RoboDK station: DK_mettoolswitch_en_meerderematen.rdk

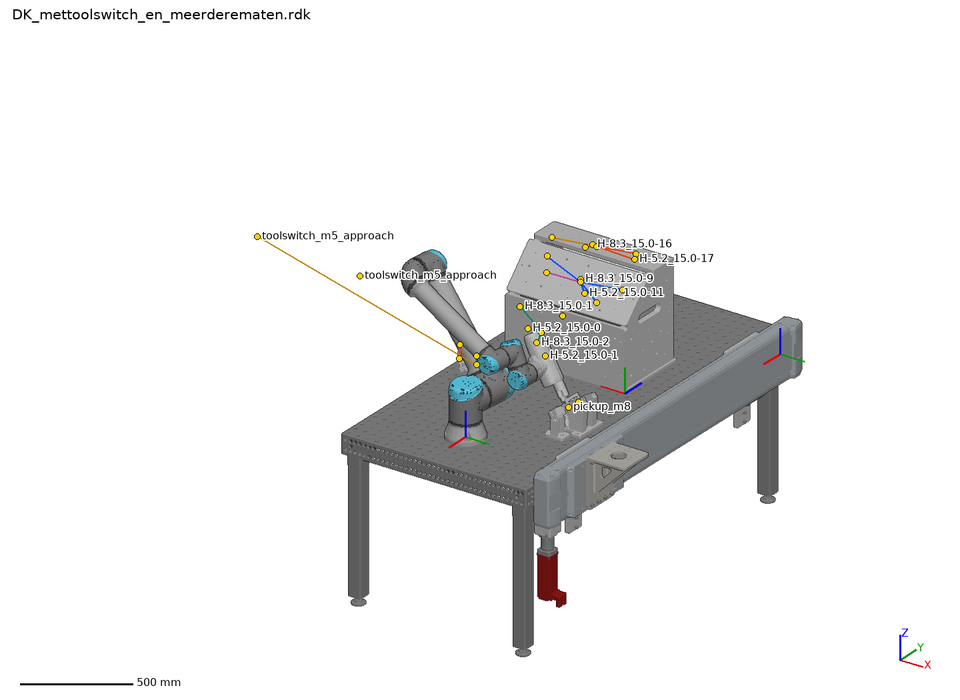
[picture v0: the station drawn from its stored meshes, robots at their saved joint values, targets as dots, program paths as lines]
Station DK_mettoolswitch_en_meerderematen (saved by RoboDK 5.9.0). Poses are relative to the parent item; angles as X-Y-Z fixed-axis rotations.
Station parameters (name, value as stored): CollisionFreePlanner, UR10e, CollisionFreePlanner-Rob UR10e, CollisionFreePlanner-Rob My Mechanism, CollisionFreePlanner-Rob Lineaire rail
  - object Lineaire Rail at (0, 0, 0) mm, size 171.1 x 1963 x 635.1 mm
  - object Cobot Carraige at (0, 0, 0) mm, size 240 x 425 x 269.5 mm
  - object Lastafel at (0, 0, 0) mm, size 1021.8 x 2000 x 842 mm
  - frame UR10e Base at (-522.25, 125.5, 70) mm, rotated rx 0 ry 0 rz -90 deg
    - robot UR10e: 6 axes, payload 10 kg, reach 1300 mm, repeatability 0.05 mm, weight 28.9 kg
        modified DH rows (alpha deg, a mm, theta deg, d mm): 0, 0, 0, 180.7; 90, 0, 180, 0; 0, 612.6, 0, 0; 0, 571.335, 0, 174.15; -90, 0, 0, 119.85; 90, 0, 180, 116.55
        joint limits [-100, -150, -30, -360, -360, -360] to [40, 0, 180, 360, 360, 360]; home [30.872, -95.296, 116.362, -22.187, 121.11, 179.827]; saved at [-96.274, -127.936, 155.823, 308.08, -8.026, -97.355]
      - tool schroevendraaier all in met nieuw kopstuk en tool, TCP at (220, -1, 100.6) mm, rotated rx 0 ry -90 rz 180 deg, size 86.2 x 139.7 x 345.9 mm, geometry from schroevendraaier all in met nieuw kopstuk en tool.STEP
  - frame Lineaire rail  Base at (218.83, 1501.27, 137) mm, rotated rx 0 ry 0 rz -90 deg
    - robot Lineaire rail: 1 axes
        modified DH rows (alpha deg, a mm, theta deg, d mm): 0, 0, 0, 0 linear
        base shift (0, 0, 0) mm, rotated rx 0 ry 90 rz 0 deg
        joint limits [-1248] to [-1248]; home [0]; saved at [-1248]
  - frame CSV Frame at (-220, 926.5, 50) mm, rotated rx 90 ry 0 rz 180 deg
    - object Test object at (0, 0, 0) mm, size 650 x 517 x 400 mm, geometry from Test object.STEP
    - object Toolswitch M5 M8 M12 (1) at (725, 0, -238) mm, size 112.6 x 60.1 x 126.6 mm, geometry from Toolswitch M5 M8 M12 (1).STEP
    - object Festo pneumatisch klem-1 at (22.5, 67, -437.5) mm, rotated rx 0 ry -90 rz -30 deg, size 249.3 x 187.1 x 198.8 mm, geometry from Festo pneumatisch klem-1.STEP
    - target pickup_m8 (Cartesian target) at (-3.8, 107.38, -439.03) mm, rotated rx 130.69 ry -86.57 rz -71.9 deg; joints [-96.274, -127.938, 155.828, 308.074, -8.028, -97.355] of UR10e
    - target pickup_m5 (Cartesian target) at (-2.38, 103.06, -363.09) mm, rotated rx 130.69 ry -86.57 rz -71.9 deg; joints [-75.565, -105.059, 145.828, -26.927, 13.754, -134.641] of UR10e
    - target H-8.3_15.0-1 (Cartesian target) at (577.65, 261.77, 15) mm; joints [-8.85, -55.871, 121.874, 293.989, -8.849, -179.992] of UR10e
    - target H-8.3_15.0-2 (Cartesian target) at (487.08, 107.86, 15) mm; joints [-11.324, -73.615, 119.159, 314.45, -11.322, -179.994] of UR10e
    - target H-8.3_15.0-9 (Cartesian target) at (325.68, 421.98, 122.91) mm, rotated rx 45 ry 0 rz 0 deg; joints [-39.434, -56.578, 53.669, 2.907, -39.433, -134.999] of UR10e
    - target H-8.3_15.0-11 (Cartesian target) at (502.06, 411.39, 112.31) mm, rotated rx 45 ry 0 rz 0 deg; joints [-28.45, -75.722, 93.025, -17.305, -28.449, -134.998] of UR10e
    - target H-8.3_15.0-16 (Cartesian target) at (391.06, 502, 308.3) mm, rotated rx -90 ry -83.43 rz 180 deg; joints [-3.833, -57.961, 69.865, -191.904, -92.74, -270.001] of UR10e
    - target H-8.3_15.0-17 (Cartesian target) at (577.65, 502, 262.67) mm, rotated rx 90 ry -81.14 rz 0 deg; joints [4.596, -59.728, 72.637, -192.908, -85.739, 89.999] of UR10e
    - target H-5.2_15.0-0 (Cartesian target) at (535.43, 162.34, 15) mm; joints [-96.274, -127.938, 155.828, 308.074, -8.028, -97.355] of UR10e
    - target H-5.2_15.0-1 (Cartesian target) at (442.81, 53.38, 15) mm; joints [-15.442, -65.401, 121.917, 303.479, -15.441, -179.996] of UR10e
    - target H-5.2_15.0-2 (Cartesian target) at (346.79, 277.43, 15) mm; joints [-24.169, -54.535, 121.923, 292.609, -24.168, -179.997] of UR10e
    - target H-5.2_15.0-10 (Cartesian target) at (534.75, 462.43, 163.36) mm, rotated rx 45 ry 0 rz 0 deg; joints [-11.699, -75.041, 88.001, 347.035, -11.697, -134.994] of UR10e
    - target H-5.2_15.0-11 (Cartesian target) at (278.01, 382.49, 83.42) mm, rotated rx 45 ry 0 rz 0 deg; joints [-11.354, -69.052, 72.632, 356.413, -11.353, -134.994] of UR10e
    - target H-5.2_15.0-12 (Cartesian target) at (103, 429.68, 130.61) mm, rotated rx 45 ry 0 rz 0 deg; joints [-31.461, -71.951, 84.687, 347.262, -31.46, -134.998] of UR10e
    - target H-5.2_15.0-15 (Cartesian target) at (197.65, 365.16, 66.09) mm, rotated rx 45 ry 0 rz 0 deg; joints [-20.089, -72.116, 80.974, 351.138, -20.088, -134.997] of UR10e
    - target H-5.2_15.0-16 (Cartesian target) at (178.59, 502, 342.35) mm, rotated rx -90 ry -85.2 rz -180 deg; joints [-17.19, -54.726, 64.672, 170.054, -77.607, -270.001] of UR10e
    - target H-5.2_15.0-17 (Cartesian target) at (151.35, 502, 290.59) mm, rotated rx 90 ry -89.07 rz 0 deg; joints [-21.263, -59.263, 71.911, 167.352, -67.807, -270.001] of UR10e
    - target H-5.2_15.0-19 (Cartesian target) at (403.31, 502, 268.12) mm, rotated rx 90 ry -77.85 rz 0 deg; joints [-7.94, -62.095, 76.272, 165.823, -69.913, -270.001] of UR10e
    - target toolswitch_m5_approach (Cartesian target) at (678.21, 67.52, -177.75) mm, rotated rx 90.07 ry 0.02 rz 0 deg; joints [-1.416, -72.071, 113.252, 318.849, -1.438, -89.956] of UR10e
      - target toolswitch_m5_approach (Cartesian target) at (678.21, 67.52, -177.75) mm, rotated rx 90.07 ry 0.02 rz 0 deg; joints [-1.416, -72.071, 113.252, 318.849, -1.438, -89.956] of UR10e
      - target toolswitch_m5_approach (Cartesian target) at (678.21, 67.52, -177.75) mm, rotated rx 90.07 ry 0.02 rz 0 deg; joints [-1.416, -72.071, 113.252, 318.849, -1.438, -89.956] of UR10e
        - target toolswitch_m5_approach (Cartesian target) at (678.21, 67.52, -177.75) mm, rotated rx 90.07 ry 0.02 rz 0 deg; joints [-1.416, -72.071, 113.252, 318.849, -1.438, -89.956] of UR10e
    - target toolswitch_m5 (Cartesian target) at (678.21, 21.65, -177.28) mm, rotated rx 90.14 ry 0.02 rz 0 deg; joints [-1.415, -68.774, 114.67, 314.195, -1.435, -89.952] of UR10e
    - target toolswitch_m8_approach (Cartesian target) at (769.79, 96.06, -177.07) mm, rotated rx 90.13 ry 0.05 rz -0.01 deg; joints [6.859, -71.505, 108.744, 322.817, 6.815, -89.924] of UR10e
    - target toolswitch_m8 (Cartesian target) at (769.77, 26.3, -177.21) mm, rotated rx 90.12 ry 0.04 rz 0 deg; joints [6.858, -66.989, 111.2, 315.836, 6.816, -89.924] of UR10e
    - target Face_Target_0 (Cartesian target) at (462.22, 165.4, 15) mm; joints [-91.475, -122.804, 153.527, 230.74, -2.975, -106.105] of UR10e
    - target Face_Target_1 (Cartesian target) at (318.87, 413.79, 114.72) mm, rotated rx 45 ry 0 rz 0 deg; joints [-91.475, -122.804, 153.527, 230.74, -2.975, -106.105] of UR10e
    - target Face_Target_2 (Cartesian target) at (364.5, 502, 302.51) mm, rotated rx -90 ry -83.43 rz 180 deg; joints [-91.475, -122.804, 153.527, 230.74, -2.975, -106.105] of UR10e
  - Python program csv_importer (listed below)
  - Python program csv_importernewest (listed below)
  - Python program Make_approaches_paths (listed below)
  - Python program TargetFixer (listed below)
  - Python program generatefaceapproaches (listed below)
  - Python program Addmoveshanktoprog (listed below)
  - Python program importerTest (listed below)
  - Python program Create measurements 3DOF (listed below)
  - Python program Prog11 (listed below)
  - Python program ProgramGenerator (listed below)
    - Python program ProgramGenerator (listed below)
  - program pickupm5Totoolswitchm8approach (13 instructions, listed below)
  - program Program_Main_Combined_met (7 instructions, listed below)
  - program Program_Main_Combined_met (13 instructions, listed below)
  - program Program_Main_Combined_met (2 instructions, listed below)
  - program Prog43 (10 instructions, listed below)
  - program pickupm8Totoolswitchm8 (12 instructions, listed below)
  - program toolswitchm8Topickupm8 (12 instructions, listed below)
  - program pickupm5Totoolswitchm5 (10 instructions, listed below)
  - program toolswitchm5Topickupm5 (10 instructions, listed below)
  - program FaceTarget0ToPickupm8 (6 instructions, listed below)
  - program Pickupm8ToFaceTarget0 (6 instructions, listed below)
  - program FaceTarget1ToPickupm8 (8 instructions, listed below)
  - program Pickupm8ToFaceTarget1 (8 instructions, listed below)
  - program FaceTarget2ToPickupm8 (15 instructions, listed below)
  - program Pickupm8ToFaceTarget2 (14 instructions, listed below)
  - program Program_Face_0_m8 (17 instructions, listed below)
  - program Program_Face_1_m8 (16 instructions, listed below)
  - program Program_Face_2_m8 (15 instructions, listed below)
  - program FaceTarget0ToPickupm5 (12 instructions, listed below)
  - program Pickupm5ToFaceTarget0 (12 instructions, listed below)
  - program FaceTarget1ToPickupm5 (12 instructions, listed below)
  - program Pickupm5ToFaceTarget1 (12 instructions, listed below)
  - program FaceTarget2ToPickupm5 (9 instructions, listed below)
  - program Pickupm5ToFaceTarget2 (8 instructions, listed below)
  - program Program_Face_0_m5 (6 instructions, listed below)
  - program Program_Face_1_m5 (33 instructions, listed below)
  - program Program_Face_2_m5 (25 instructions, listed below)
  - program Program_Main_m8 (5 instructions, listed below)
  - program Program_Main_m5 (5 instructions, listed below)
  - program pickupm8Totoolswitchm8approach (16 instructions, listed below)
  - program toolswitchm8approachTopickupm8 (16 instructions, listed below)
  - program Tool_Pickup_m8 (5 instructions, listed below)
  - program Tool_Dropoff_m8 (5 instructions, listed below)
  - program pickupm5Totoolswitchm5approach (12 instructions, listed below)
  - program toolswitchm5approachTopickupm5 (12 instructions, listed below)
  - program Tool_Pickup_m5 (6 instructions, listed below)
  - program Tool_Dropoff_m5 (5 instructions, listed below)
  - program Program_Main_Combined (8 instructions, listed below)
  - program toolswitchm5approachTopickupm8 (13 instructions, listed below)
  - program pickupm8Totoolswitchm5approach (13 instructions, listed below)
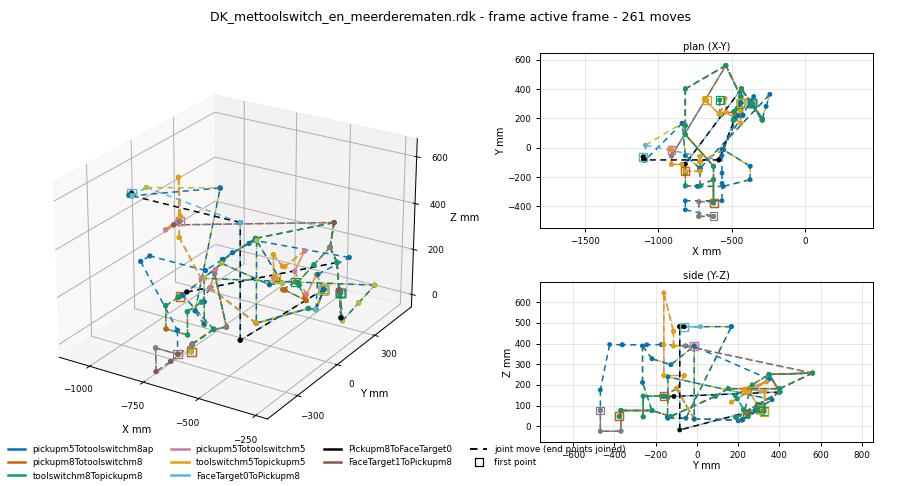
[picture p0: tool path of DK_mettoolswitch_en_meerderematen.rdk in frame active frame, 261 of 322 moves have a stored position in this frame; points joined in program order, loops and branches not executed]
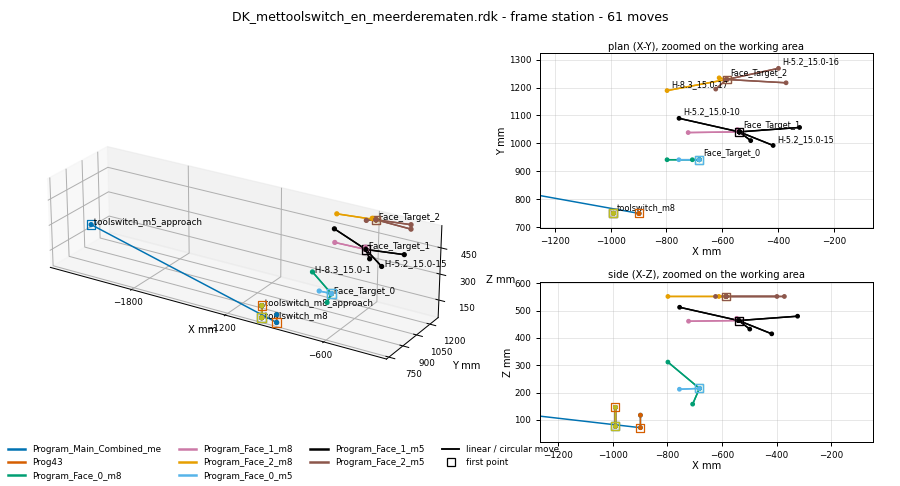
[picture p1: tool path of DK_mettoolswitch_en_meerderematen.rdk in frame station, 61 of 322 moves have a stored position in this frame; points joined in program order, loops and branches not executed]

--- Python program csv_importer ---
# This macro can load CSV files from Denso programs in RoboDK.
# Supported types of files are:
#  1-Tool data : Tool.csv
#  2-Work object data: Work.csv
#  3-Target data: P_Var.csv
# This macro can also filter a given targets file

# Type help("robodk.robolink") or help("robodk.robomath") for more information
# Press F5 to run the script
# Visit: http://www.robodk.com/doc/PythonAPI/
# For RoboDK API documentation

import os
import datetime

import tkinter as tk
from tkinter import messagebox

from robodk.robolink import *  # API to communicate with RoboDK
from robodk.robomath import *  # Robot toolbox
from robodk.robodialogs import *
from robodk.robofileio import *
import robodk.robolinkutils as RDKutils

DEBUG = False

debuglist = []

# Start communication with RoboDK
RDK = Robolink()

# Ask the user to select the robot
ROBOT = RDK.ItemUserPick('Select a robot', ITEM_TYPE_ROBOT)

# Check if the user selected a robot
if not ROBOT.Valid():
    quit()


# Ask the user to select a reference frame and get the active tool
BASE = ROBOT.Parent()
#BASE = RDK.Item('UR10e Base', ITEM_TYPE_FRAME)
#BASE = RDK.ItemUserPick('Select robot base frame', ITEM_TYPE_FRAME)
FRAME = RDK.ItemUserPick('Reference Frame', ITEM_TYPE_FRAME)
FRAMEPOSE = RDKutils.getPoseWrt(FRAME, BASE) #frame pose wrt robot base
TOOL = ROBOT.getLink(ITEM_TYPE_TOOL)
TOOLPOSE = RDKutils.getPoseWrt(TOOL, TOOL.Parent()) #tool pose wrt robot flange

if not FRAME.Valid() or not TOOL.Valid():
    raise Exception("Select appropriate FRAME and TOOL references")


# Function to convert XYZWPR to a pose
# Important! Specify the order of rotation
def xyzwpr_to_pose(xyzwpr):
    x, y, z, rx, ry, rz = xyzwpr
    return point_Zaxis_2_pose([x, y, z], [-rx, -ry, -rz])



# csv_file = 'C:/Users/Albert/Desktop/Var_P.csv'
csv_file = getOpenFileName(RDK.getParam('PATH_OPENSTATION'))

# Specify file codec
codec = 'utf-8'  #'ISO-8859-1'

def mirror_target(xyzwpr):
    """
    Mirrors the target position and adjusts the rotation.
    Assumes the wall is aligned with the YZ plane (mirroring the X coordinate).
    """
    x, y, z, rx, ry, rz = xyzwpr

    # Mirror the position (reflect across the YZ plane)
    x_mirrored = x  # Negate the X coordinate
    y_mirrored = y   # Keep Y and Z the same
    z_mirrored = z

    # Adjust the rotation (flip RX and RZ)
    rx_mirrored = rx  # Negate RX
    ry_mirrored = ry   # Keep RY the same
    rz_mirrored = -rz  # Negate RZ

    return [x_mirrored, y_mirrored, z_mirrored, rx_mirrored, ry_mirrored, rz_mirrored]

def load_targets(strfile):
    csvdata = LoadList(strfile, ',', codec)
    poses = []
    idxs = []
    for i in range(0, len(csvdata)):
        x, y, z, rx, ry, rz = csvdata[i][0:6]

        # Mirror the target
        x_mirrored, y_mirrored, z_mirrored, rx_mirrored, ry_mirrored, rz_mirrored = mirror_target([x, y, z, rx, ry, rz])

        # Convert the mirrored target to a pose
        poses.append(xyzwpr_to_pose([x_mirrored, y_mirrored, z_mirrored, rx_mirrored, ry_mirrored, rz_mirrored]))
        idxs.append(i)
    return poses, idxs


# Load and display Targets from P_Var.CSV in RoboDK
def make_targets(strfile):
    """Load and display Targets from P_Var.CSV in RoboDK with robust error handling."""
    # Initialize empty lists to collect results
    poses, idxs = load_targets(strfile)
    program_name = getFileName(strfile)
    program_name = program_name.replace('-', '_').replace(' ', '_')

    holes_no_solution = []
    total_targets = len(poses)
    processed_targets = 0

    # Show progress message
    RDK.ShowMessage(f"Processing {total_targets} targets...", False)

    # Process each target
    for pose, idx in zip(poses, idxs):
        try:
            processed_targets += 1
            if processed_targets % 5 == 0:  # Update progress every 5 targets
                RDK.ShowMessage(f"Processing target {processed_targets} of {total_targets}...", False)

            name = 'H-%s-%i' % (program_name, idx)

            # Check if target already exists and delete it
            target = RDK.Item(name, ITEM_TYPE_TARGET)
            if target.Valid():
                target.Delete()

            # Create new target and set pose
            target = RDK.AddTarget(name, FRAME, ROBOT)
            target.setPose(pose)

            # Try to find a collision-free configuration
            if not find_collision_free_configuration(target, idx):
                holes_no_solution.append(idx)
                if DEBUG:
                    print(f"No solution for Hole {idx}")
                    debuglist.append(f"No solution for Hole {idx}")

        except Exception as e:
            # Log error but continue with next target
            holes_no_solution.append(idx)
            if DEBUG:
                print(f"Error processing Hole {idx}: {e}")
                debuglist.append(f"Error processing Hole {idx}: {e}")

    # Show completion message
    if holes_no_solution:
        RDK.ShowMessage(f"Completed with {len(holes_no_solution)} targets without solution: {holes_no_solution}", False)
    else:
        RDK.ShowMessage("All targets processed successfully!", False)

    return holes_no_solution

def test_collision_safe(pose, test_move=False):
    """
    Test a pose for collisions without triggering script interruption.

    Args:
        pose: The pose to test
        test_move: Whether to actually move the robot (False = calculate only)

    Returns:
        0: No collision detected
        1: Collision detected
        -2: Pose unreachable
    """
    # Turn off collision detection while we test
    RDK.setCollisionActive(COLLISION_OFF)

    try:
        # Check if the pose is reachable without moving
        joints = ROBOT.SolveIK(pose, TOOLPOSE, FRAMEPOSE)

        if joints is None or len(joints) == 0:
            return -2  # Unreachable

        if test_move:
            # Try moving to the position with collisions off
            try:
                ROBOT.MoveJ(joints)
            except:
                return -2  # Problem moving, treat as unreachable

        # Check collision after positioning but without movement
        # This allows us to check without triggering interruption
        RDK.setCollisionActive(COLLISION_ON)
        collision = RDK.Collisions()

        if collision > 0:
            return 1  # Collision detected
        else:
            return 0  # No collision

    except Exception as e:
        if DEBUG:
            print(f"Error in collision testing: {e}")
            debuglist.append(f"Error in collision testing: {e}")
        return -2  # Any error, treat as unreachable

    finally:
        # Always make sure we turn collision checking back off
        RDK.setCollisionActive(COLLISION_OFF)


def test_all_configurations(configurations):
    """Test all robot configurations and find one without collisions.
    Returns:
        0: If a collision-free configuration is found
        1: If all configurations have collisions
        -2: If no configurations are reachable
    """
    if not configurations:
        return -2  # No configurations available

    for joints in configurations:
        # Turn collision checking off for movement
        RDK.setCollisionActive(COLLISION_OFF)

        # Try to move to target configuration with error handling
        try:
            ROBOT.MoveJ(joints)
        except Exception as e:
            if DEBUG:
                print(f"Error moving to configuration: {e}")
                debuglist.append(f"Error moving to configuration: {e}")
            continue  # Skip this configuration

        # Check for collisions without moving
        try:
            RDK.setCollisionActive(COLLISION_ON)
            collision = RDK.Collisions()

            # If no collision, we found a valid configuration
            if collision == 0:
                return 0

        except Exception as e:
            if DEBUG:
                print(f"Error checking collision: {e}")
                debuglist.append(f"Error checking collision: {e}")
            continue  # Skip this configuration on error

    # All configurations had issues
    return 1

def test_collision_target(target):
    """
    Test if the current target pose is collision-free.
    Optimized to quickly check multiple configurations.
    """
    try:
        if DEBUG:
            print("Testing target for collisions")
            debuglist.append("Testing target for collisions")

        # Get all possible configurations for this target
        possible_configurations = ROBOT.SolveIK_All(target.Pose(), tool=TOOLPOSE, reference=FRAMEPOSE)

        # Quick check - if no configurations are possible, fail early
        if not possible_configurations or len(possible_configurations) == 0:
            return -2

        # Test configurations in batches for efficiency
        return test_all_configurations(possible_configurations)

    except Exception as e:
        if DEBUG:
            print(f"Error in test_collision_target: {e}")
            debuglist.append(f"Error in test_collision_target: {e}")
        return 1  # Assume collision on error

def test_issues_point(target, rz):
    if DEBUG:
        print("testing point")
        debuglist.append("testing point")

    # define the rotated position to test for collisions
    target_new_pose = RelTool(target.Pose(), 0,0,0, 0,0,rz)
    possible_robot_configurations = ROBOT.SolveIK_All(target_new_pose, tool=TOOLPOSE, reference=FRAMEPOSE)
    issues_value = test_all_configurations(possible_robot_configurations) # returns 0 if at least one configuration is without issues

    return issues_value, target_new_pose

rotation_direction = "pos"
direction_changes = 0
holes_no_solution = []

def find_collision_free_configuration(target, idx):
    """
    Find a collision-free configuration for the target by trying different rotations.
    This version avoids script interruption on collision detection.

    Returns:
        True if a collision-free configuration was found, False otherwise
    """
    # Store original pose to restore if needed
    original_pose = target.Pose()

    # First check if original pose is collision-free
    result = test_collision_safe(original_pose)
    if result == 0:
        if DEBUG:
            print(f"Original pose for Hole {idx} is collision-free")
            debuglist.append(f"Original pose for Hole {idx} is collision-free")
        return True

    # Define rotation search strategy
    # Use an incremental approach rather than testing all at once
    rotation_axes = ['z', 'y', 'x']  # Order matters - most likely axis first
    angles_to_try = [15, 30, 45, 60, 90, 120, 150, 180, -15, -30, -45, -60, -90, -120, -150, -180]

    # Track best rotation setup
    best_result = 1  # 1 = collision, we want 0 = no collision
    best_pose = None

    # Try each axis and angle combination
    for axis in rotation_axes:
        for angle in angles_to_try:
            try:
                # Create a new rotated pose
                if axis == 'z':
                    new_pose = RelTool(original_pose, 0, 0, 0, 0, 0, angle)
                elif axis == 'y':
                    new_pose = RelTool(original_pose, 0, 0, 0, 0, angle, 0)
                elif axis == 'x':
                    new_pose = RelTool(original_pose, 0, 0, 0, angle, 0, 0)

                # Test this pose
                result = test_collision_safe(new_pose)

                # If collision-free, we can use this one
                if result == 0:
                    if DEBUG:
                        print(f"Found collision-free pose for Hole {idx} with {axis} rotation of {angle}")
                        debuglist.append(f"Found collision-free pose for Hole {idx} with {axis} rotation of {angle}")

                    # Set the target pose and return success
                    target.setPose(new_pose)
                    return True

                # Update best result if this is better
                if result < best_result:
                    best_result = result
                    best_pose = new_pose

            except Exception as e:
                if DEBUG:
                    print(f"Error testing {axis} rotation of {angle} for Hole {idx}: {e}")
                    debuglist.append(f"Error testing {axis} rotation of {angle} for Hole {idx}: {e}")

    # If we get here, no completely collision-free pose was found
    # If we found a feasible but colliding pose, use that as a fallback
    if best_pose is not None:
        try:
            target.setPose(best_pose)
            if DEBUG:
                print(f"Using best available pose for Hole {idx} (not collision-free)")
                debuglist.append(f"Using best available pose for Hole {idx} (not collision-free)")
        except:
            # If setting pose fails, restore original
            target.setPose(original_pose)
    else:
        # Restore original pose
        target.setPose(original_pose)

    if DEBUG:
        print(f"No collision-free pose found for Hole {idx}")
        debuglist.append(f"No collision-free pose found for Hole {idx}")

    return False

def rotate_target(pose, axis, angle):
    """Rotate target pose around specified axis by given angle."""
    try:
        if axis.lower() == 'z':
            return RelTool(pose, 0, 0, 0, 0, 0, angle)
        elif axis.lower() == 'y':
            return RelTool(pose, 0, 0, 0, 0, angle, 0)
        elif axis.lower() == 'x':
            return RelTool(pose, 0, 0, 0, angle, 0, 0)
        else:
            return pose
    except Exception as e:
        if DEBUG:
            print(f"Error rotating target ({axis}, {angle}): {e}")
            debuglist.append(f"Error rotating target ({axis}, {angle}): {e}")
        return pose



def main():
    global holes_no_solution
    holes_no_solution = []

    MAKE_GUI_PROGRAM = True

    ROBOT.setFrame(FRAME)
    ROBOT.setTool(TOOL)

    if RDK.RunMode() == RUNMODE_SIMULATE:
        MAKE_GUI_PROGRAM = True
    else:
        MAKE_GUI_PROGRAM = False

    if MAKE_GUI_PROGRAM:
        # Disable rendering for speed
        RDK.Render(False)

        # Process the targets
        holes_no_solution = make_targets(csv_file)

        # Re-enable rendering
        RDK.Render(True)

        # Final report
        if holes_no_solution:
            final_message = f"Completed with {len(holes_no_solution)} holes without solution: {holes_no_solution}"
            RDK.ShowMessage(final_message, False)
            if DEBUG:
                print(final_message)
                debuglist.append(final_message)

                # Write debug info to file
                current_time = datetime.datetime.now()
                filename = os.path.splitext(os.path.basename(__file__))
                with open("debugfile.txt", "a") as file:
                    file.write("\n\n-----------------------------------------------\n")
                    file.write(current_time.strftime("%c"))
                    file.write("\n-----------------------------------------------\n")
                    for prints in debuglist:
                        file.write(str(prints))
                        file.write("\n")
                    file.write(str(holes_no_solution))
                    file.write(str(filename[0]))

# Run the main function
if __name__ == "__main__":
    main()
else:
    main()  # For RoboDK compatibility, run even if imported

--- Python program csv_importernewest ---
# This macro can load CSV files from Denso programs in RoboDK.
# Supported types of files are:
#  1-Tool data : Tool.csv
#  2-Work object data: Work.csv
#  3-Target data: P_Var.csv
# This macro can also filter a given targets file

# Type help("robodk.robolink") or help("robodk.robomath") for more information
# Press F5 to run the script
# Visit: http://www.robodk.com/doc/PythonAPI/
# For RoboDK API documentation

import os
import datetime

import tkinter as tk
from tkinter import messagebox

from robodk.robolink import *  # API to communicate with RoboDK
from robodk.robomath import *  # Robot toolbox
from robodk.robodialogs import *
from robodk.robofileio import *
import robodk.robolinkutils as RDKutils

DEBUG = False

debuglist = []

# Start communication with RoboDK
RDK = Robolink()

# Ask the user to select the robot
ROBOT = RDK.ItemUserPick('Select a robot', ITEM_TYPE_ROBOT)

# Check if the user selected a robot
if not ROBOT.Valid():
    quit()


# Ask the user to select a reference frame and get the active tool
BASE = ROBOT.Parent()
#BASE = RDK.Item('UR10e Base', ITEM_TYPE_FRAME)
#BASE = RDK.ItemUserPick('Select robot base frame', ITEM_TYPE_FRAME)
FRAME = RDK.ItemUserPick('Reference Frame', ITEM_TYPE_FRAME)
FRAMEPOSE = RDKutils.getPoseWrt(FRAME, BASE) #frame pose wrt robot base
TOOL = ROBOT.getLink(ITEM_TYPE_TOOL)
TOOLPOSE = RDKutils.getPoseWrt(TOOL, TOOL.Parent()) #tool pose wrt robot flange

if not FRAME.Valid() or not TOOL.Valid():
    raise Exception("Select appropriate FRAME and TOOL references")


# Function to convert XYZWPR to a pose
# Important! Specify the order of rotation
def xyzwpr_to_pose(xyzwpr):
    x, y, z, rx, ry, rz = xyzwpr
    return point_Zaxis_2_pose([x, y, z], [-rx, -ry, -rz])
    #return transl(x, y, z) * rotz(rz * pi / 180) * roty(ry * pi / 180) * rotx(rx * pi / 180)
    #return transl(x,y,z)*rotx(rx*pi/180)*roty(ry*pi/180)*rotz(rz*pi/180)
    #return KUKA_2_Pose(xyzwpr)


# csv_file = 'C:/Users/Albert/Desktop/Var_P.csv'
csv_file = getOpenFileName(RDK.getParam('PATH_OPENSTATION'))

# Specify file codec
codec = 'utf-8'  #'ISO-8859-1'


# Load P_Var.CSV data as a list of poses, including links to reference and tool frames
def load_targets(strfile):
    csvdata = LoadList(strfile, ',', codec)
    poses = []
    idxs = []
    for i in range(0, len(csvdata)):
        x, y, z, rx, ry, rz = csvdata[i][0:6]
        poses.append(xyzwpr_to_pose([x, y, z, rx, ry, rz]))
        #idxs.append(csvdata[i][6])
        idxs.append(i)

    return poses, idxs


# Load and display Targets from P_Var.CSV in RoboDK
def make_targets(strfile):
    poses, idxs = load_targets(strfile)
    program_name = getFileName(strfile)
    program_name = program_name.replace('-', '_').replace(' ', '_')

    for pose, idx in zip(poses, idxs):
        name = 'H-%s-%i' % (program_name, idx)
        target = RDK.Item(name, ITEM_TYPE_TARGET)
        if target.Valid():
            target.Delete()
        target = RDK.AddTarget(name, FRAME, ROBOT)


        target.setPose(pose)
        collision_free(target, idx)

def test_all_configurations(configurations):
    for joints in configurations:

        # turn collision checking off
        RDK.setCollisionActive(COLLISION_OFF)

        # move to target
        try:
            ROBOT.MoveJ(joints)
        except TargetReachError:
            continue

        # turn collision checking on, test for collisions
        RDK.setCollisionActive(COLLISION_ON)

        collision = RDK.Collisions()
        print(f"collision: {collision}")
        debuglist.append(f"collision: {collision}")

        collision_items = RDK.CollisionItems()
        if TOOL in collision_items or collision == 0:
            break

    try:
        collision
    except NameError:
        collision = -2
        print("Target cannot be reached or is to close to a singularity")
        debuglist.append("Target cannot be reached or is to close to a singularity")

    return collision


def test_collision_target(target, rz):
    if DEBUG:
        print("testing at target")
        debuglist.append("testing at target")

    possible_robot_configurations = ROBOT.SolveIK_All(target.Pose(), tool=TOOLPOSE, reference=FRAMEPOSE)
    issues_value = test_all_configurations(possible_robot_configurations) # returns 0 if at least one configuration is without issues

    return issues_value

def test_issues_point(target, rz, flip_approach=False):
    if DEBUG:
        print("testing point")
        debuglist.append("testing point")

    # Get the original pose
    original_pose = target.Pose()

    # For vertical walls, we might need to completely flip the approach
    if flip_approach:
        # Rotate 180 degrees around Y axis (assuming Y is the axis parallel to the wall)
        # This effectively approaches from the opposite direction
        target_new_pose = RelTool(original_pose, 0, 0, 0, 0, 180, 0)
        # Then apply the requested Z rotation
        target_new_pose = RelTool(target_new_pose, 0, 0, 0, 0, 0, rz)
    else:
        # Standard rotation around Z axis only
        target_new_pose = RelTool(original_pose, 0, 0, 0, 0, 0, rz)

    possible_robot_configurations = ROBOT.SolveIK_All(target_new_pose, tool=TOOLPOSE, reference=FRAMEPOSE)
    issues_value = test_all_configurations(possible_robot_configurations)

    return issues_value, target_new_pose

rotation_direction = "pos"
direction_changes = 0
holes_no_solution = []

def collision_free(target, idx):
    rotation_step = 30
    repmax = 360/rotation_step
    global rotation_direction
    global direction_changes
    s = 0
    rep = 0

    print(f"\nHole {idx}")
    debuglist.append(f"\nHole {idx}")

    # First try the original approach
    issues_value, target_new_pose = test_issues_point(target, 0, flip_approach=False)

    # If there's a collision, try different approaches
    while issues_value != 0 and s < 100:
        print(f"s before: {s}")
        debuglist.append(f"s before: {s}")
        print(f"rep: {rep}")
        debuglist.append(f"rep: {rep}")
        print(f"rotation direction: {rotation_direction}")
        debuglist.append(f"rotation direction: {rotation_direction}")
        print(f"direction changes: {direction_changes}")
        debuglist.append(f"direction changes: {direction_changes}")

        s += 1

        # For unreachable targets or potential vertical wall collision situations
        if issues_value == -2 and direction_changes < 2:
            if rotation_direction == "pos":
                rotation_direction = "neg"
                direction_changes += 1
                r = -1
            else:
                rotation_direction = "pos"
                direction_changes += 1
                r = 1

            # Try the opposite approach direction if we've changed direction once already
            # This is key for vertical walls
            if direction_changes >= 1:
                issues_value, target_new_pose = test_issues_point(target, r*rotation_step, flip_approach=True)
            else:
                issues_value, target_new_pose = test_issues_point(target, r*rotation_step, flip_approach=False)

            target.setPose(target_new_pose)

        # For collision situations, rotate around Z
        elif issues_value > 0 and rep < repmax:
            RDK.setCollisionActive(COLLISION_OFF) # collision off

            ROBOT.MoveJ(target.Pose())

            if rotation_direction == "neg":
                r = -1
            elif rotation_direction == "pos":
                r = 1

            # After trying several rotations, try the flip approach
            if rep > repmax/2:
                issues_value, target_new_pose = test_issues_point(target, r*rotation_step, flip_approach=True)
            else:
                issues_value, target_new_pose = test_issues_point(target, r*rotation_step, flip_approach=False)

            target.setPose(target_new_pose)
            rep += 1

        elif direction_changes >= 2 or rep >= repmax:
            break

        else:
            RDK.ShowMessage(f"Unknown error occured at Hole {idx} while looking for collision free position")

    direction_changes = 0
    if issues_value == 0:
        print(f"No issues at Hole {idx}")
        debuglist.append(f"No issues at Hole {idx}")
    elif direction_changes >= 2 or rep >= repmax or s >= 100:
        RDK.ShowMessage(f"No solution found for Hole {idx}", False)
        holes_no_solution.append(idx)

        print(f"No solution found for Hole {idx}")
        debuglist.append(f"No solution found for Hole {idx}")

    else:
        RDK.ShowMessage(f"Unknown error occured at Hole {idx} while looking for collision free position")

        print(f"Unknown error occured at Hole {idx} while looking for collision free position")
        debuglist.append(f"Unknown error occured at Hole {idx} while looking for collision free position")


MAKE_GUI_PROGRAM = True

ROBOT.setFrame(FRAME)
ROBOT.setTool(TOOL)

if RDK.RunMode() == RUNMODE_SIMULATE:
    MAKE_GUI_PROGRAM = True
    # MAKE_GUI_PROGRAM = mbox('Do you want to create a new program? If not, the robot will just move along the targets', 'Yes', 'No')
else:
    # if we run in program generation mode just move the robot
    MAKE_GUI_PROGRAM = False

if MAKE_GUI_PROGRAM:
    RDK.Render(False)  # Faster if we turn render off
    make_targets(csv_file)
else:
    l

if len(holes_no_solution) != 0:
    RDK.ShowMessage(f"Holes without solution: {holes_no_solution}")

if DEBUG:
    print(f"Holes without solution: {holes_no_solution}")
    debuglist.append(f"Holes without solution: {holes_no_solution}")

    current_time = datetime.datetime.now()
    filename = os.path.splitext(os.path.basename(__file__))
    with open("C:/Users/Laura/Documents/1.Windesheim/Stage/2024/Lectoraat/Deelvragen/2.Targets maken/debugfile.txt", "a") as file:
        file.write("\n\n-----------------------------------------------\n")
        file.write(current_time.strftime("%c"))
        file.write("\n-----------------------------------------------\n")
        for prints in debuglist:
            file.write(prints)
            file.write("\n")
        file.write(holes_no_solution)
        file.write(filename[0])

--- Python program Make_approaches_paths ---
from robodk.robolink import *  # API to communicate with RoboDK
from robodk.robomath import *  # Robot toolbox
import robodk.robolinkutils as RDKutils


DEBUG = False


# Link to RoboDK
RDK = Robolink()

ROBOT = RDK.ItemUserPick('Select a Robot', ITEM_TYPE_ROBOT)
FRAME = RDK.ItemUserPick('Reference Frame', ITEM_TYPE_FRAME)

if not ROBOT.Valid() or not FRAME.Valid():
    raise Exception("Select appropriate ROBOT and FRAME")

BASE = RDK.Item('UR10e Base', ITEM_TYPE_FRAME)
#BASE = RDK.ItemUserPick('Select robot base frame', ITEM_TYPE_FRAME)
FRAMEPOSE = RDKutils.getPoseWrt(FRAME, BASE) #frame pose wrt robot base
TOOL = ROBOT.getLink(ITEM_TYPE_TOOL)
TOOLPOSE = RDKutils.getPoseWrt(TOOL, TOOL.Parent()) #tool pose wrt robot flange




# get all the holes as items
All_items = RDK.ItemList(ITEM_TYPE_TARGET)
#RDK_items = [item for item in All_items if "Hole" in item.Name()]
RDK_items = [item for item in All_items if "H" in item.Name()]
print(f"Holes: {len(RDK_items)}")

RDK.setCollisionActive(COLLISION_OFF)

def print_xyzrpw(pose):
    x, y, z, rx, ry, rz = pose_2_xyzrpw(pose)
    print(x, y, z, rx, ry, rz)


class Hole:
    def __init__(self, pose, target):
        self.pose = pose
        self.target = target
        self.name = self.target.Name()
        self.split_position_rotation(pose)

    def split_position_rotation(self, pose):
        x, y, z, rx, ry, rz = pose_2_xyzrpw(pose)
        self.position = x, y, z
        # get the way the z-axis is facing
        self.rotation = pose[0:3,2] # from all 3 rows (0:3) only the 3rd column (index 2) (the last column of the rotation matrix)
        # format the z-axis facing, so it can be made a key in the dictonary
        zfacing1 = round(self.rotation.tolist()[0])
        zfacing2 = round(self.rotation.tolist()[1])
        zfacing3 = round(self.rotation.tolist()[2])
        self.rot_identifier = f"{zfacing1}_{zfacing2}_{zfacing3}"

class Face:
    def __init__(self, key):
        self.key = key
        self.get_midpoint(key)
        self.rotation = self.holes[0].rotation.tolist()
        self.offset_multiplier = self.rotation
        self.approaches = []

    def get_midpoint(self, key):
        #global dic
        #targets from key
        self.holes = dic[key]
        #x, y, z from targets
        self.x_values = []
        self.y_values = []
        self.z_values = []
        for hole in self.holes:
            x, y, z = hole.position
            self.x_values.append(x)
            self.y_values.append(y)
            self.z_values.append(z)
        if DEBUG:
            print("ranges:")
            print(self.x_values)
            print(self.y_values)
            print(self.z_values)
        #min and max of these
        self.x_values.sort()
        min_x = self.x_values[0]
        max_x = self.x_values[len(self.x_values)-1]
        offset_x = (max_x - min_x)/2
        mid_x = max_x - offset_x
        self.xranges = min_x, max_x, mid_x

        self.y_values.sort()
        min_y = self.y_values[0]
        max_y = self.y_values[len(self.y_values)-1]
        offset_y = (max_y - min_y)/2
        mid_y = max_y - offset_y
        self.yranges = min_y, max_y, mid_y

        self.z_values.sort()
        min_z = self.z_values[0]
        max_z = self.z_values[len(self.z_values)-1]
        offset_z = (max_z - min_z)/2
        mid_z = max_z - offset_z
        self.zranges = min_z, max_z, mid_z

        self.midpoint = mid_x, mid_y, mid_z

        self.ref_hole = self.holes[0]
        ref_pose = self.ref_hole.pose
        ref_pose[0,3] = mid_x
        ref_pose[1,3] = mid_y
        ref_pose[2,3] = mid_z
        self.midpose = ref_pose
        if DEBUG:
            print("min, max, mid: ")
            print("x: ", self.xranges)
            print("y: ", self.yranges)
            print("z: ", self.zranges)
            print("midpoint: ", self.midpoint)
            print("midpose: ", self.midpose)

    def add_approaches(self, approach):
        self.approaches.append(approach)



class Approach:
    def __init__(self, face, number):
        self.face = face
        self.number = number
        self.target = self.make_approach_target(face, number)

    def make_approach_target(self, face, number):
        approach_point = self.get_approach_point(face)
        approach_target = RDK.Item(f"approach {idx} {face.rotation}", ITEM_TYPE_TARGET)
        if approach_target.Valid():
            approach_target.Delete()
        approach_target = RDK.AddTarget(f"approach {idx} {face.rotation}", FRAME, ROBOT)
        approach_target.setPose(approach_point)
        if DEBUG:
            print("approach target:\n", approach_point)
        return approach_target

    def get_approach_point(self, face):
        MAX_APPROACH = 100 #in mm
        MIN_APPROACH = 20 #in mm
        STEP = 40 #in mm
        ROT_STEP = 20 #in degrees
        approach_point = self.test_distance(face, MAX_APPROACH, MIN_APPROACH, STEP, ROT_STEP)
        return approach_point

    def test_distance(self, face, MAX_APPROACH, MIN_APPROACH, STEP, ROT_STEP):
        approach_distance = MAX_APPROACH
        rep = 0
        repmax = 360/ROT_STEP
        rot_offset = 0
        rotation_direction = "pos"
        direction_changes = 0

        z = approach_distance
        issues, approach_point = self.test_point(face.midpose, z, 0)
        #first_issues_value = issues
        if issues == -2:
            rz = 180
            rot_offset = rz
            issues, approach_point = self.test_point(face.midpose, z, rz)

        sa = 0
        while issues != 0 and approach_distance >= MIN_APPROACH + STEP and sa < 100:
            sa += 1
            approach_distance -= STEP
            z = approach_distance
            rz = 0
            issues, approach_point = self.test_point(face.midpose, z, rz)
            issues, approach_point = self.rotate(face, issues, approach_distance, rot_offset, ROT_STEP)

        return approach_point

    def rotate(self, face, issues, approach_distance, rot_offset, ROT_STEP):
        repmax = 360/ROT_STEP
        rotation_direction = "pos"
        direction_changes = 0
        rep = 0
        sb = 0
        while issues != 0 and sb < 100:
            sb += 1
            if issues == -2 and direction_changes < 2:
                if rotation_direction == "pos":
                    rotation_direction = "neg"
                    r = -1 #rotation factor to make the rotation negative
                else:
                    rotation_direction = "pos"
                    r = 1
                direction_changes += 1
                z = approach_distance
                rz = rot_offset + r * ROT_STEP
                issues, approach_point = self.test_point(face.midpose, z, rz)
            elif issues > 0 and rep < repmax:
                if rotation_direction == "neg":
                    r = -1
                else:
                    r = 1
                rep += 1
                z = approach_distance
                rz = rot_offset + r * ROT_STEP
                rot_offset = rz
                issues, approach_point = self.test_point(face.midpose, z, rz)
            elif direction_changes >= 2 or rep >= repmax:
                break

            else:
                print(f"Unknown error occured at Approach {self.number}")

        if issues != 0 and (direction_changes >= 2 or rep >= repmax or sb == 100):
            print(f"No solution found for Approach {self.number}")
            global approach_noSolution
            approach_noSolution.append(self.number)
            RDK.ShowMessage(f"No solution found for Approach {self.number}", False)
        return issues, approach_point

    def test_point(self, point, z, rz):
        # define the position to test for collisions
        test_point = RelTool(point, 0,0,z, 0,0,rz)
        possible_robot_configurations = ROBOT.SolveIK_All(test_point, tool=TOOLPOSE, reference=FRAMEPOSE)
        issues = self.test_all_configurations(possible_robot_configurations)
        return issues, test_point

    def test_all_configurations(self, configurations):
        for joints in configurations:

            # turn collision checking off
            RDK.setCollisionActive(COLLISION_OFF)
            is_active = RDK.Command("CollisionActive")
            #print(f"collsion active? should be off (0) {is_active}")

            # move to target
            try:
                ROBOT.MoveJ(joints)
            except TargetReachError:
                continue

            # turn collision checking on, test for collisions
            RDK.setCollisionActive(COLLISION_ON)
            is_active = RDK.Command("CollisionActive")
            #print(f"collsion active? should be on (1) {is_active}")
            collision = RDK.Collisions()
            #print(f"collision: {collision}")
            collision_items = RDK.CollisionItems()
            if TOOL in collision_items or collision == 0:
                break

        try:
            collision
        except NameError:
            collision = -2 # TargetReachError occures for every configuration
            #print("Target cannot be reached or is to close to a singularity")

        return collision

def collision_free_paths(face, approach):
    possible_configurations = ROBOT.SolveIK_All(approach.target.Pose(), tool=TOOLPOSE, reference=FRAMEPOSE)
    for i, joints in enumerate(possible_configurations):
        print(f"testing configuration {i+1}")
        for j, hole in enumerate(face.holes):
            RDK.setCollisionActive(COLLISION_OFF)
            ROBOT.MoveJ(joints)
            RDK.setCollisionActive(COLLISION_ON)
            issues = ROBOT.MoveJ_Test(joints, hole.target.Joints())
            print(f"Hole {hole.name} with issues = {issues}")
            if issues == 0:
                continue
            break

        if issues == 0:
            print(f"found valid configuration: {i+1}")
            approach.target.setJoints(joints)
            break

    if issues != 0:
        print(f"no configuration found for approach {approach.number}")
        path_no_solution.append(hole.name)

holes = []
dic = {}
faces = []
approach_noSolution = []
path_no_solution = []

# convert the target items into target objects
for item in RDK_items:
    hole = Hole(item.Pose(), item)
    holes.append(hole)

# put the targets with the z-axis facing the same way together
for hole in holes:
    if hole.rot_identifier in dic:
        #dic exists put it in
        dic[hole.rot_identifier].append(hole)
    else:
        #make a dic and put it in
        dic[hole.rot_identifier] = [hole]

keys = list(dic.keys())
for key in keys:
    if DEBUG:
        print(f"{key}: {dic[key]}")
    face = Face(key)
    faces.append(face)
    if DEBUG:
        print(face.midpoint)

for idx, face in enumerate(faces):
    if DEBUG:
        print(faces)
    approach = Approach(face, idx)
    face.add_approaches(approach)

    #paden maken tussen approach en targets die daar bij horen
    for approach in face.approaches:
        collision_free_paths(face, approach)
        for hole in face.holes:
            program_name = f"to {hole.name}"
            program = RDK.Item(program_name, ITEM_TYPE_PROGRAM)
            if program.Valid():
                program.Delete()
            program = RDK.AddProgram(program_name, ROBOT)
            ROBOT.MoveJ(approach.target)
            program.MoveJ(hole.target)

--- Python program TargetFixer ---
from robodk import robolink, robomath
import robodk.robolinkutils as RDKutils

from robodk.robolink import *       # RoboDK API
from robodk.robomath import *        # Math toolbox (provides transl, etc.)
from robodk.robodialogs import *
from robodk.robofileio import *

def main():
    # Initialize RoboDK instance
    RDK = robolink.Robolink()

    # Let the user pick a Robot and a Reference Frame
    ROBOT = RDK.ItemUserPick('Select a Robot', ITEM_TYPE_ROBOT)
    FRAME = RDK.ItemUserPick('Select a Reference Frame', ITEM_TYPE_FRAME)
    if not ROBOT.Valid() or not FRAME.Valid():
        raise Exception("Select appropriate ROBOT and FRAME")

    # Get Base, Tool and FRAME pose (adjust names as needed)
    BASE = RDK.Item('UR10e Base', ITEM_TYPE_FRAME)
    FRAMEPOSE = RDKutils.getPoseWrt(FRAME, BASE) if BASE.Valid() else FRAME.Pose()
    TOOL = ROBOT.getLink(ITEM_TYPE_TOOL)
    TOOLPOSE = RDKutils.getPoseWrt(TOOL, TOOL.Parent())

    # Activate collision checking
    RDK.setCollisionActive(COLLISION_ON)

    # Get all targets (or filter them as needed)
    all_targets = RDK.ItemList(ITEM_TYPE_TARGET)

    fixed_targets = []
    unfixed_targets = []

    # Process every target one by one
    for target in all_targets:
        original_pose = target.Pose()
        print(f"\nProcessing target: {target.Name()}")

        # First, check if the target is already collision free:
        if not target_in_collision(RDK, ROBOT, target, FRAMEPOSE, TOOLPOSE):
            print(f"Target {target.Name()} is already collision free. No fix needed.")
            continue

        print(f"Target {target.Name()} is in collision. Attempting to fix by shifting along principal axes...")

        # Try to fix by shifting along X, then Y, then Z
        fixed = fix_target(target, original_pose, RDK, ROBOT, FRAMEPOSE, TOOLPOSE)
        if fixed:
            fixed_targets.append(target.Name())
        else:
            unfixed_targets.append(target.Name())
            target.setPose(original_pose)  # revert to original if no fix was found

    # Summary report
    print("\nTarget fixing complete.")
    print("Fixed targets:")
    for t in fixed_targets:
        print("  -", t)
    if unfixed_targets:
        print("Targets that could not be fixed:")
        for t in unfixed_targets:
            print("  -", t)

def target_in_collision(RDK, ROBOT, target, FRAMEPOSE, TOOLPOSE):
    """
    Checks whether the given target causes a collision.
    It does so by attempting to solve IK and simulating a MoveJ.
    Returns True if a collision (or no valid configuration) is detected.
    """
    pose = target.Pose()
    possible_configs = ROBOT.SolveIK_All(pose, tool=TOOLPOSE, reference=FRAMEPOSE)
    if not possible_configs:
        return True
    for joints in possible_configs:
        try:
            ROBOT.MoveJ(joints)
        except Exception:
            continue
        if not RDK.Collisions():
            return False
    return True

def fix_target(target, original_pose, RDK, ROBOT, FRAMEPOSE, TOOLPOSE):
    """
    Attempts to fix a target by shifting it along each principal axis.

    For each axis (X, Y, Z), the function:
      - Tries a positive shift in 10-mm increments (10 steps).
      - Reverts to the original pose.
      - Tries a negative shift in 10-mm increments (10 steps).

    If a collision-free pose is found during any of these tests, the target is updated.
    Returns True if a valid pose is found, otherwise False.
    """
    # Define axes along which to shift using lambda functions that generate translation matrices.
    # The transl(x, y, z) function creates a translation matrix in the local coordinate system when multiplied with a pose.
    axes = [
        ("X", lambda d: transl(d, 0, 0)),
        ("Y", lambda d: transl(0, d, 0)),
        ("Z", lambda d: transl(0, 0, d))
    ]

    # For each axis...
    for axis_name, shift_func in axes:
        # Try positive direction shifts first
        for i in range(1, 11):
            shift_matrix = shift_func(10 * i)  # 10-mm increments
            test_pose = original_pose * shift_matrix
            target.setPose(test_pose)
            if not target_in_collision(RDK, ROBOT, target, FRAMEPOSE, TOOLPOSE):
                print(f"Target {target.Name()} fixed with a +{10*i} mm shift along {axis_name}.")
                return True
        # Revert to the original pose before trying the negative direction
        target.setPose(original_pose)
        for i in range(1, 11):
            shift_matrix = shift_func(-10 * i)
            test_pose = original_pose * shift_matrix
            target.setPose(test_pose)
            if not target_in_collision(RDK, ROBOT, target, FRAMEPOSE, TOOLPOSE):
                print(f"Target {target.Name()} fixed with a {-10*i} mm shift along {axis_name}.")
                return True
        # Revert to the original pose before trying the next axis
        target.setPose(original_pose)
    return False

if __name__ == '__main__':
    main()

--- Python program generatefaceapproaches ---
from robodk.robolink import *  # API to communicate with RoboDK
from robodk.robomath import *   # Robot toolbox
import robodk.robolinkutils as RDKutils
from robodk import robolink

DEBUG = False

# Link to RoboDK
RDK = Robolink()

ROBOT = RDK.ItemUserPick('Select a Robot', ITEM_TYPE_ROBOT)
FRAME = RDK.ItemUserPick('Reference Frame', ITEM_TYPE_FRAME)

if not ROBOT.Valid() or not FRAME.Valid():
    raise Exception("Select appropriate ROBOT and FRAME")

BASE = RDK.Item('UR10e Base', ITEM_TYPE_FRAME)
FRAMEPOSE = RDKutils.getPoseWrt(FRAME, BASE)  # frame pose with respect to robot base
TOOL = ROBOT.getLink(ITEM_TYPE_TOOL)
TOOLPOSE = RDKutils.getPoseWrt(TOOL, TOOL.Parent())  # tool pose with respect to robot flange

# Get all the holes as targets (only those with "H" in the name)
All_items = RDK.ItemList(ITEM_TYPE_TARGET)
RDK_items = [item for item in All_items if "H" in item.Name()]
print(f"Holes: {len(RDK_items)}")

RDK.setCollisionActive(COLLISION_OFF)

def print_xyzrpw(pose):
    x, y, z, rx, ry, rz = pose_2_xyzrpw(pose)
    print(x, y, z, rx, ry, rz)

class Hole:
    def __init__(self, pose, target):
        self.pose = pose
        self.target = target
        self.name = self.target.Name()
        self.split_position_rotation(pose)

    def split_position_rotation(self, pose):
        x, y, z, rx, ry, rz = pose_2_xyzrpw(pose)
        self.position = (x, y, z)
        # Get the z-axis direction (3rd column of the rotation matrix)
        self.rotation = pose[0:3, 2]
        zfacing1 = round(self.rotation.tolist()[0])
        zfacing2 = round(self.rotation.tolist()[1])
        zfacing3 = round(self.rotation.tolist()[2])
        self.rot_identifier = f"{zfacing1}_{zfacing2}_{zfacing3}"

class Face:
    def __init__(self, key):
        self.key = key
        self.get_midpoint(key)
        self.rotation = self.holes[0].rotation.tolist()
        self.offset_multiplier = self.rotation
        self.approaches = []  # Not used in the new functions

    def get_midpoint(self, key):
        # Retrieve all holes corresponding to this face
        self.holes = dic[key]
        x_values = [hole.position[0] for hole in self.holes]
        y_values = [hole.position[1] for hole in self.holes]
        z_values = [hole.position[2] for hole in self.holes]

        # Sort and compute the midpoint as the average of the min and max values
        x_values.sort()
        y_values.sort()
        z_values.sort()
        min_x, max_x = x_values[0], x_values[-1]
        min_y, max_y = y_values[0], y_values[-1]
        min_z, max_z = z_values[0], z_values[-1]

        mid_x = (min_x + max_x) / 2
        mid_y = (min_y + max_y) / 2
        mid_z = (min_z + max_z) / 2

        self.midpoint = (mid_x, mid_y, mid_z)

        # Use the first hole's pose as a template and update its translation to the midpoint
        self.ref_hole = self.holes[0]
        ref_pose = self.ref_hole.pose
        ref_pose[0, 3] = mid_x
        ref_pose[1, 3] = mid_y
        ref_pose[2, 3] = mid_z
        self.midpose = ref_pose

    def add_approaches(self, approach):
        self.approaches.append(approach)

# --- Process holes and group them into faces based on z-axis orientation ---
holes = []
dic = {}
faces = []

# Convert the target items into Hole objects
for item in RDK_items:
    hole = Hole(item.Pose(), item)
    holes.append(hole)

# Group holes with the same z-axis orientation (rounded)
for hole in holes:
    if hole.rot_identifier in dic:
        dic[hole.rot_identifier].append(hole)
    else:
        dic[hole.rot_identifier] = [hole]

# Create Face objects from the groups
for key in dic:
    face = Face(key)
    faces.append(face)

# --- NEW FUNCTION: Create face targets at the midpoint of each face ---
def create_face_targets():
    """
    For each computed face, create a new target in RoboDK at the face midpoint.
    """
    for i, face in enumerate(faces):
        face_target_name = f"Face_Target_{i}"

        # Delete existing target if it exists
        existing_target = RDK.Item(face_target_name, ITEM_TYPE_TARGET)
        if existing_target.Valid():
            existing_target.Delete()

        # Start with the original midpose
        collision_free_pose = face.midpose.copy()
        collision_found = True

        print(f"Checking collision for face {i} at midpoint {face.midpoint}")

        # Enable collision detection
        RDK.setCollisionActive(COLLISION_ON)

        # First try the original pose (0 degrees)
        ROBOT.setPose(face.midpose)
        collision = RDK.Collisions()

        if collision == 0:
            collision_free_pose = face.midpose
            collision_found = False
            print(f"Found collision-free pose for face {i} with rz = 0 degrees")
        else:
            # Try alternating positive and negative rotations
            rotation_step = 10
            max_rotation = 720

            while collision_found and rotation_step <= max_rotation:
                # Try both positive and negative rotations for this step
                for rotation_direction in ["pos", "neg"]:
                    if rotation_direction == "neg":
                        r = -1
                    elif rotation_direction == "pos":
                        r = 1

                    rz = r * rotation_step
                    test_pose = RelTool(face.midpose, 0, 0, 0, 0, 0, rz)

                    # Set robot to test pose and check for collision
                    ROBOT.setPose(test_pose)
                    collision = RDK.Collisions()

                    if collision == 0:
                        # No collision found - we can use this pose
                        collision_free_pose = test_pose
                        collision_found = False
                        print(f"Found collision-free pose for face {i} with rz = {rz} degrees")
                        break
                    else:
                        print(f"Collision detected for face {i} at rz = {rz}, continuing search...")

                # If collision-free pose found, break out of the while loop
                if not collision_found:
                    break

                # Increment rotation step for next iteration
                rotation_step += 10

        if collision_found:
            print(f"Warning: Could not find collision-free pose for face {i} after full rotation (±{max_rotation}°)")
            # Use original pose anyway
            collision_free_pose = face.midpose

        # Create the face target with the collision-free pose
        face_target = RDK.AddTarget(face_target_name, FRAME, ROBOT)
        face_target.setPose(collision_free_pose)

        print(f"Created face target for face {i} at midpoint {face.midpoint}")

    # Turn off collision detection when done
    RDK.setCollisionActive(COLLISION_OFF)



# --- NEW FUNCTION: Create a program for each face using MoveL commands ---
def create_face_programs():
    """
    For each face, generate a program that moves from the face target (approach target)
    to every hole target on that face using a MoveL command.
    Each move from the face target to a hole target is followed by a return move to the face target.
    """

    for i, face in enumerate(faces):
        face_target_name = f"Face_Target_{i}"
        face_target = RDK.Item(face_target_name, ITEM_TYPE_TARGET)
        prog_name = f"Program_Face_{i}"
        existing_prog = RDK.Item(prog_name, ITEM_TYPE_PROGRAM)
        if existing_prog.Valid():
            existing_prog.Delete()
        prog = RDK.AddProgram(prog_name, ROBOT)

        # Add a move to the face target as the starting (approach) move


        # For each hole in this face, add a MoveL to go to the hole target and then a MoveL back to the face target.
        for j, hole in enumerate(face.holes):  # Use enumerate to get the index 'j' of the hole

            # Construct the program names using f-strings
            program_to_call_2 = f'pickupToFaceTarget{i}'
            program_to_call_1 = f'FaceTarget{i}Topickup'

            if j == 0:
                prog.RunInstruction(program_to_call_2, robolink.INSTRUCTION_CALL_PROGRAM)

            prog.MoveL(face_target)
            prog.MoveL(hole.target)

            prog.RunInstruction('screw_in(20)', robolink.INSTRUCTION_CALL_PROGRAM)  # Tighten screw
            prog.RunInstruction('screw_out(0)', robolink.INSTRUCTION_CALL_PROGRAM)  # Release screwdriver

            prog.MoveL(face_target)

            prog.RunInstruction(program_to_call_1, robolink.INSTRUCTION_CALL_PROGRAM)

            # Check if it's NOT the last hole in the face
            if j < len(face.holes) - 1:

                prog.RunInstruction(program_to_call_2, robolink.INSTRUCTION_CALL_PROGRAM)

            print(f"Program {prog_name}: Added MoveL from approach target to hole {hole.name} and back.")

def addmainprogram():


    prog_name = f"Program_Main"
    existing_prog = RDK.Item(prog_name, ITEM_TYPE_PROGRAM)
    if existing_prog.Valid():
        existing_prog.Delete()
    prog = RDK.AddProgram(prog_name, ROBOT)


    # set reference frame
    # set tcp
    prog.setTool(RDK.ItemUserPick('Select tool', ITEM_TYPE_TOOL))
    prog.setFrame(RDK.ItemUserPick('Select frame', ITEM_TYPE_FRAME))

    # Voeg elke program toe aan een groot programma die met "program_face" begint
    for j in range(len(faces)):
        sub_prog_name = f"Program_Face_{j}"
        prog.RunInstruction(sub_prog_name)



def generate_pickup_links():

    # for i, face in enumerate(faces):
    #     ROBOT.setPoseFrame(face.midpose[i]) ## deze lijn
    #     status = RDK.PluginCommand("CollisionFreePlanner", "Add")
    #     print(status)

    # Define the name that is given in RoboDK for the pickup target
    pickup_target_name = "pickup"  # The name of the target in your RoboDK station

    # Get the actual RoboDK Item for the pickup target
    Target_Pickup_item = RDK.Item(pickup_target_name, ITEM_TYPE_TARGET)

    if not Target_Pickup_item.Valid():
        print(
            f"Error: Pickup target '{pickup_target_name}' not found in RoboDK station. Skipping pickup link generation.")
        return  # Exit the function if the pickup target doesn't exist

    # For every face, create 2 planned motions (programs)
    # One from Face_Target_i to 'pickup' target
    # One from 'pickup' target to Face_Target_i
    for i, face in enumerate(faces):  # Iterate through faces to get the numerical index 'i'
        # Get the name of the Face_Target for the current face
        face_target_name = f"Face_Target_{i}"

        # Define the names for the programs to be created by the plugin
        program_name_to_pickup = f"FaceTarget{i}Topickup"
        program_name_from_pickup = f"pickupToFaceTarget{i}" # Corrected: consistency with previous example

        # --- Check and delete existing "To Pickup" program ---
        existing_prog_to_pickup = RDK.Item(program_name_to_pickup, ITEM_TYPE_PROGRAM)
        if existing_prog_to_pickup.Valid():
            print(f"Deleting existing program: {program_name_to_pickup}")
            existing_prog_to_pickup.Delete()

        print(f"Attempting to join: {face_target_name} to {pickup_target_name} as {program_name_to_pickup}")

        # Call the plugin command to join the face target to the pickup target
        status_to_pickup = RDK.PluginCommand(
            "CollisionFreePlanner",
            "Join",
            f"{face_target_name}|{pickup_target_name}|{program_name_to_pickup}"
            )
        print(f"Status for '{program_name_to_pickup}': {status_to_pickup}")

        # --- Check and delete existing "From Pickup" program ---
        existing_prog_from_pickup = RDK.Item(program_name_from_pickup, ITEM_TYPE_PROGRAM)
        if existing_prog_from_pickup.Valid():
            print(f"Deleting existing program: {program_name_from_pickup}")
            existing_prog_from_pickup.Delete()

        print(f"Attempting to join: {pickup_target_name} to {face_target_name} as {program_name_from_pickup}")

        # Call the plugin command to join the pickup target to the face target
        status_from_pickup = RDK.PluginCommand(
            "CollisionFreePlanner",
            "Join",
            f"{pickup_target_name}|{face_target_name}|{program_name_from_pickup}"
             )
        print(f"Status for '{program_name_from_pickup}': {status_from_pickup}")


    print("\nPickup link generation process finished.")

#def generate_unscrewing_programs():


# --- Main execution: Run only the new functions ---
if __name__ == '__main__':
    create_face_targets()
    generate_pickup_links()
    create_face_programs()
    addmainprogram()

#for documentation of the collision free motion planner see https://robodk.com/addin/com.robodk.plugin.collisionfreeplanner, searched ages for API documentation

--- Python program Addmoveshanktoprog ---
from robodk import robolink, robomath

# Connect to RoboDK
RDK = robolink.Robolink()

# Ask the user to select the program to duplicate
orig_prog = RDK.ItemUserPick("Select the program to duplicate", robolink.ITEM_TYPE_PROGRAM)
if not orig_prog.Valid():
    print("No valid program selected.")
    quit()

# Create a new program (a duplicate) with a new name
new_prog_name = "New_" + orig_prog.Name()
new_prog = RDK.AddProgram(new_prog_name)
print("Creating new program:", new_prog.Name())

# Get the number of instructions from the original program
ins_count = orig_prog.InstructionCount()
print("Original program '{}' has {} instructions.".format(orig_prog.Name(), ins_count))

# Iterate over each instruction in the original program
for i in range(ins_count):
    # Retrieve instruction info as a dictionary.
    # Note: Calling setParam(i) with only the index returns the instruction information.
    ins_dict = orig_prog.setParam(i)

    # Try to get the command code string from the instruction dictionary.
    # (Many instructions have a "Code" key that holds the Python command as text.)
    code_line = ins_dict.get("Code", "").strip()
    if not code_line:
        print("Skipping instruction {} because no code is available.".format(i))
        continue

    # Add the instruction to the new program
    print("Adding instruction {}: {}".format(i, code_line))
    new_prog.RunInstruction(code_line, robolink.INSTRUCTION_CALL_PROGRAM)

    # If the instruction contains "FaceTarget" then add two extra moveshank instructions after it.
    if "Face_Target" in code_line:
        print("Detected 'FaceTarget' at instruction {}. Inserting moveshank instructions.".format(i))
        new_prog.RunInstruction('move_shank(20)', robolink.INSTRUCTION_CALL_PROGRAM)
        new_prog.RunInstruction('move_shank(0)', robolink.INSTRUCTION_CALL_PROGRAM)

# Finalize the new program; this applies the modifications
new_prog.Update()
print("New program '{}' created successfully.".format(new_prog.Name()))

--- Python program importerTest ---
# This macro loads CSV target files and places them in RoboDK
# Supported CSV format: X,Y,Z,RX,RY,RZ

# Import required modules
from robodk.robolink import *  # API to communicate with RoboDK
from robodk.robomath import *  # Robot toolbox
from robodk.robodialogs import *
from robodk.robofileio import *
import robodk.robolinkutils as RDKutils

# Start communication with RoboDK
RDK = Robolink()

# Ask the user to select the robot
ROBOT = RDK.ItemUserPick('Select a robot', ITEM_TYPE_ROBOT)

# Check if the user selected a robot
if not ROBOT.Valid():
    quit()

# Get the reference frame and active tool
BASE = ROBOT.Parent()
FRAME = RDK.ItemUserPick('Reference Frame', ITEM_TYPE_FRAME)
FRAMEPOSE = RDKutils.getPoseWrt(FRAME, BASE)  # frame pose wrt robot base
TOOL = ROBOT.getLink(ITEM_TYPE_TOOL)
TOOLPOSE = RDKutils.getPoseWrt(TOOL, TOOL.Parent())  # tool pose wrt robot flange

if not FRAME.Valid() or not TOOL.Valid():
    raise Exception("Select appropriate FRAME and TOOL references")

# Function to convert XYZWPR to a pose
def xyzwpr_to_pose(xyzwpr):
    x, y, z, rx, ry, rz = xyzwpr
    return point_Zaxis_2_pose([x, y, z], [rx, ry, rz])

# Ask user to select the CSV file
csv_file = getOpenFileName(RDK.getParam('PATH_OPENSTATION'))

# Specify file codec
codec = 'utf-8'

# Load CSV target data
def load_targets(strfile):
    csvdata = LoadList(strfile, ',', codec)
    poses = []
    idxs = []
    for i in range(0, len(csvdata)):
        x, y, z, rx, ry, rz = csvdata[i][0:6]
        poses.append(xyzwpr_to_pose([x, y, z, rx, ry, rz]))
        idxs.append(i)
    return poses, idxs

# Create targets in RoboDK and move the robot to each target
def process_targets(strfile):
    poses, idxs = load_targets(strfile)
    program_name = getFileName(strfile)
    program_name = program_name.replace('-', '_').replace(' ', '_')

    # Set the robot's frame and tool
    ROBOT.setFrame(FRAME)
    ROBOT.setTool(TOOL)

    # Create a program to visit all targets
    program = RDK.AddProgram('Visit_' + program_name, ROBOT)

    for pose, idx in zip(poses, idxs):
        # Create target name
        name = 'Target-%s-%i' % (program_name, idx)

        # Delete target if it already exists
        target = RDK.Item(name, ITEM_TYPE_TARGET)
        if target.Valid():
            target.Delete()

        # Create new target
        target = RDK.AddTarget(name, FRAME, ROBOT)
        target.setPose(pose)

        # Add a movement instruction to the program
        program.MoveJ(target)

        # Optional: Move the robot to the target in simulation
        RDK.setSimulationSpeed(1)  # Normal speed
        ROBOT.MoveJ(target)

# Main execution
if __name__ == "__main__":
    # Ask user whether to just create targets or also move the robot
    move_robot = RDK.RunMode() != RUNMODE_SIMULATE

    if move_robot:
        # We're in run mode, just move the robot to targets
        poses, idxs = load_targets(csv_file)
        for pose, idx in zip(poses, idxs):
            ROBOT.MoveJ(pose)
    else:
        # We're in simulation mode, create targets and a program
        process_targets(csv_file)

    RDK.ShowMessage("Target processing complete", False)

--- Python program Create measurements 3DOF ---
# type help("robolink") or help("robodk") for more information
# (note: you do not need to keep a copy of this file, your python script is saved with the station)
from robodk.robolink import *  # API to communicate with robodk
from robodk.robomath import *  # basic matrix operations
from robodk.robodialogs import *
from random import uniform
import sys  # to exit the script without errors (sys.exit(0))
import re  # to convert a string list into a list of values


def CreateMeasurementsPoint(calib_targets=None):

    DEFAULT_NMEASURES = 80
    # Default limit space in the Cartesian space
    DEFAULT_XYZ_MIN = [-5000, -5000, 0]
    DEFAULT_XYZ_MAX = [5000, 5000, 5000]

    TRACKER_REF_NAME = 'Tracker Reference'  # keyword of the measurement system reference (in RoboDK)
    TCP_PREFIX = 'CalibTool'

    # Use the tag CHECK_COLLISION_NAME to automatically turn the objects visible. This will allow to detect collisions.
    CHECK_COLLISION = True
    CHECK_COLLISION_MOVE = True
    CHECK_COLLISION_NAME = 'collision'
    CHECK_COLLISION_STEP = -1  # in degrees, step to check for collisions. higher is faster.

    # Use the tag CHECK_COLLISION_NAME to automatically turn the objects visible. This will allow to detect collisions.
    CHECK_WORKSPACE = False
    CHECK_WORKSPACE_NAME = 'Workspace'

    # Avoid a cylinder located at X=0, Y=0 or radius R_MIN
    R_MIN = 100
    R_MIN_Z = 200

    # Allow rotations of the tool pointing to the measurement system
    ROTX_MIN = -5
    ROTX_MAX = 5
    ROTY_MIN = -5
    ROTY_MAX = 5
    ROTZ_MIN = -180
    ROTZ_MAX = 180

    # use FILE_SAVE_PREFIX to automatically save the file, otherwise, comment this line
    # FILE_SAVE_PREFIX = 'CalibrationSequence'

    # --------------------------------------------------------------
    def to_list(str_values, expected_values):
        """Converts a string into a list of values. It returns None if the array is smaller than the expected size."""
        if str_values is None:
            return None
        values = re.findall("[-+]?\d+[\.]?\d*", str_values)
        if len(values) < expected_values:
            return None
        for i in range(len(values)):
            values[i] = float(values[i])
        print('Read values: ' + repr(values))
        return values

    def get_values(title_msg, show_value, expected_values):
        """Gets a list of values from the user, stops the script if the user hits cancel"""
        if type(show_value) == Mat:
            show_value = show_value.tolist()
        answer = mbox(title_msg, entry=str(show_value))
        if answer is False:
            print('Operation cancelled by user')
            sys.exit(0)
            #raise Exception('Operation cancelled by user')
        #print('Input value: ' + answer)
        values = to_list(answer, expected_values)
        #if len(values) < expected_values:
        #    raise Exception('%i values expected' % expected_values)
        return values

    def stop_script():
        """Forces the script to finish with/without errors"""
        # raise Exception('Operation cancelled by user')
        print('Operation cancelled by user')
        sys.exit(0)

    # ---------------------------------
    RDK = Robolink()

    # Disable collision checking (otherwise, the program stops)
    RDK.setCollisionActive(COLLISION_OFF)

    # get previously set variables
    NMEASURES = RDK.getParam('CALIB_MEASUREMENTS')
    #JOINTS_REF = to_list(RDK.getParam('CALIB_JOINTS_REF'), 6)
    ANG_MIN = to_list(RDK.getParam('CALIB_JOINTLIM_LOW'), 6)
    ANG_MAX = to_list(RDK.getParam('CALIB_JOINTLIM_HIGH'), 6)
    XYZ_MIN = to_list(RDK.getParam('CALIB_XYZLIM_LOW'), 3)
    XYZ_MAX = to_list(RDK.getParam('CALIB_XYZLIM_HIGH'), 3)

    INPUT_VALUES = False
    # force user input if one of the variables is not set
    if NMEASURES is None or ANG_MIN is None or ANG_MAX is None:  # or XYZ_MIN is None or XYZ_MAX is None:
        INPUT_VALUES = True

    #----------------------- Select robot ------------------
    robot = RDK.ItemUserPick("Select a robot for calibration/validation", ITEM_TYPE_ROBOT)
    if not robot.Valid():
        raise Exception('Robot not selected or no robot available')
    print('Using robot: %s' % robot.Name())
    #------------------------------------------------------------

    #----------------------- Select tracker ------------------
    tracker = RDK.Item(TRACKER_REF_NAME)
    if not tracker.Valid():
        frame_ref = RDK.AddFrame('Measurements Reference', robot.Parent())
        frame_ref.setPose(transl(2000, 0, 1000))
        tracker = RDK.AddFrame(TRACKER_REF_NAME, frame_ref)
        tracker.setPose(transl(0, 0, 0))
        tracker.setVisible(False)
    #    tracker = RDK.ItemUserPick('Select the measurement system reference:<br>(avoid this message by naming the tracker reference "%s")' % TRACKER_REF_NAME, ITEM_TYPE_FRAME)
    #    if not tracker.Valid():
    #        stop_script()

    #----------------------- Select tool and workspace object to verify if tool is inside the object
    tool_object = None
    workspace_object = None
    if CHECK_WORKSPACE:
        # tool_object is the geometry of the tool used to check if the tool is inside the workspace
        robot_tools = robot.Childs()
        for tooli in robot_tools:
            if tooli.Name().find(CHECK_COLLISION_NAME) >= 0:
                tool_object = tooli
        if tool_object is None and len(robot_tools) > 0:
            tool_object = robot_tools[0]

        # workspace object is the workspace of the tracker (object)
        workspace_object = RDK.Item(CHECK_WORKSPACE_NAME, ITEM_TYPE_OBJECT)
    #------------------------------------------------------------

    #if JOINTS_REF is None:
    #    # Use robot home position as default reference joints
    #    JOINTS_REF = robot.JointsHome().tolist()

    if XYZ_MIN is None:
        XYZ_MIN = DEFAULT_XYZ_MIN

    if XYZ_MAX is None:
        XYZ_MAX = DEFAULT_XYZ_MAX

    [ang_min_robot, ang_max_robot, JOINTS_TYPE] = robot.JointLimits()
    if ANG_MIN is None or ANG_MAX is None:
        ANG_MIN = ang_min_robot.tolist()
        ANG_MAX = ang_max_robot.tolist()
        # limit joint axes from -180 to +180 (no need to go farther for calibration)
        for i in [3, 5]:
            ANG_MIN[i] = max(ANG_MIN[i], -180)
            ANG_MAX[i] = min(ANG_MAX[i], 180)

        ANG_MIN[0] = max(ANG_MIN[0], -90)
        ANG_MAX[0] = min(ANG_MAX[0], 90)

        ANG_MIN[4] = max(ANG_MIN[4], -90)
        ANG_MAX[4] = min(ANG_MAX[4], 90)

        print('Using default robot joint limits:')
        print(ANG_MIN)
        print(ANG_MAX)

    while True:
        # Loop until the user inputs variables that are accepted
        if INPUT_VALUES:
            # Ask the user to validate/enter all the settings

            # ---------------- getting the number of measurements
            if NMEASURES is None or type(NMEASURES) == str:
                NMEASURES = DEFAULT_NMEASURES
            input_val = mbox('Enter the number of measurements:\n(at least 60 measurements are recommended for robot calibration)', entry=str(NMEASURES))
            if input_val is False:
                stop_script()

            NMEASURES = int(float(input_val))
            RDK.setParam('CALIB_MEASUREMENTS', NMEASURES)

            # ---------------- getting the Reference Joints
            #robot.setJoints(JOINTS_REF)
            #answer = mbox('Set the robot reference joints and select OK. The tool must be facing the tracker for this position.\nCurrent values: %s' % str(JOINTS_REF))
            #if answer is False:
            #    stop_script()

            #JOINTS_REF = robot.Joints().tolist()
            #RDK.setParam('CALIB_JOINTS_REF', JOINTS_REF)

            # ---------------- getting the Joint limits (lower bound)
            robot.setJoints(ANG_MIN)
            answer = mbox('Set the Joint limits (LOWER bound, in deg), then select OK.\nCurrent values: %s' % str(ANG_MIN))
            if answer is False:
                stop_script()

            ANG_MIN = robot.Joints().tolist()
            RDK.setParam('CALIB_JOINTLIM_LOW', ANG_MIN)

            # ---------------- getting the Joint limits (upper bound)
            robot.setJoints(ANG_MAX)
            answer = mbox('Set the Joint limits (UPPER bound, in deg), then select OK.\nCurrent values: %s' % str(ANG_MAX))
            if answer is False:
                stop_script()

            ANG_MAX = robot.Joints().tolist()
            RDK.setParam('CALIB_JOINTLIM_HIGH', ANG_MAX)

            # ---------------- getting the XYZ limits (lower bound)
            #XYZ_MIN = get_values('Enter the Cartesian limits (lower bound, in mm), then select OK.', XYZ_MIN, 3)
            #RDK.setParam('CALIB_XYZLIM_LOW', XYZ_MIN)

            # ---------------- getting the XYZ limits (upper bound)
            #XYZ_MAX = get_values('Enter the Cartesian limits (upper bound, in mm), then select OK.', XYZ_MAX, 3)
            #RDK.setParam('CALIB_XYZLIM_HIGH', XYZ_MAX)

        # show summary of parameters
        #robot.setJoints(JOINTS_REF)
        summary_msg = 'Current settings to generate robot calibration configurations:\n\n'
        summary_msg += ('Number of points: %i\n' % NMEASURES)
        #summary_msg += ('Reference joints (deg): %s\n' % str([ round(elem) for elem in JOINTS_REF ]))
        summary_msg += ('Tracker object: %s\n' % tracker.Name())
        if tool_object is not None and workspace_object is not None and workspace_object.Valid() and workspace_object.Visible():
            CHECK_WORKSPACE = True
            summary_msg += ('Creating targets inside tracker workspace (hide workspace to deactivate)\n\n')
        else:
            CHECK_WORKSPACE = False
            summary_msg += ('Skip creating targets inside the tracker workspace (show workspace to activate)\n\n')
        summary_msg += ('Lower joint limits (deg): %s\n' % str(ANG_MIN))
        summary_msg += ('Upper joint limits (deg): %s\n\n' % str(ANG_MAX))
        summary_msg += ('Lower Cartesian limits (mm): %s\n' % str(XYZ_MIN))
        summary_msg += ('Upper Cartesian limits (mm): %s\n\n' % str(XYZ_MAX))
        summary_msg += ('Important: Define collision map settings to check for collisions (select: Tools->Collision Map)\n\n')
        summary_msg += ('Continue?')

        answer = mbox(summary_msg, b1=('Start', 's'), b2=('Edit', 'e'))
        pause(0.001)  # Make tkinter disappear on Mac
        if answer == 'e':
            # Continue loop until the summary is accepted
            INPUT_VALUES = True
            continue

        # if paramters are OK, exit the loop and continue
        break

    # raise Exception('done')

    NDOFS = min(len(robot.Joints().list()), len(ANG_MAX))

    # -----------------------------------------------------
    # Custom-made procedures
    def randjoints():
        """Returns a random set of robot joints within the joint limits."""
        angrand = Mat(NDOFS, 1)
        for i in range(NDOFS):
            angrand[i, :] = uniform(ANG_MIN[i], ANG_MAX[i])
        #jrand = angles_2_joints(angrand.tolist(), JOINTS_TYPE)
        jrand = angrand.tolist()
        return Mat(jrand)

    def check_joints(jin):
        """Returns true if the joints are within the accepted limits."""
        if not isinstance(jin, Mat):
            return False
        if jin.size(0) < 6:
            return False
        #angles = joints_2_angles(jin.tolist(), JOINTS_TYPE)
        angles = jin.tolist()
        for i in range(NDOFS):
            if angles[i] > ANG_MAX[i] or angles[i] < ANG_MIN[i]:
                print("        Joint %i out of limits (%.1f)" % ((i + 1), angles[i]))
                return False
        return True

    def check_pose(hin):
        """Returns true if the pose is within the accepted limits."""
        x = hin[0, 3]
        y = hin[1, 3]
        z = hin[2, 3]
        if x < XYZ_MIN[0] or x > XYZ_MAX[0]:
            print("        X coordinate out of limits %.1f" % x)
        elif y < XYZ_MIN[1] or y > XYZ_MAX[1]:
            print("        Y coordinate out of limits %.1f" % y)
        elif z < XYZ_MIN[2] or z > XYZ_MAX[2]:
            print("        Z coordinate out of limits %.1f" % z)
        elif x * x + y * y < R_MIN * R_MIN and z < R_MIN_Z:
            print("        Robot wrist too close to the robot")
        else:
            return True
        return False

    def randpose(rob, htool, point):
        """Returns a random pose where the Z axis points to the measurement system within the accepted rotation limits.
        The point must be given with respect to the robot reference frame."""
        while True:
            jrand = randjoints()
            try:
                print("Random joints: " + str(jrand.list()))
                hrand = rob.SolveFK(jrand) * htool
            except:
                continue
            prand = hrand[0:3, 3].tolist()
            zvect = normalize3(subs3(point, prand))
            xaprox = [0, 0, 1]
            if angle3(zvect, xaprox) < 5 * pi / 180:
                xaprox = [0, 1, 0]
            yvect = normalize3(cross(zvect, xaprox))
            xvect = cross(yvect, zvect)
            hrand[0:3, 0] = xvect
            hrand[0:3, 1] = yvect
            hrand[0:3, 2] = zvect
            rx = uniform(ROTX_MIN, ROTX_MAX) * pi / 180
            ry = uniform(ROTY_MIN, ROTY_MAX) * pi / 180
            rz = uniform(ROTZ_MIN, ROTZ_MAX) * pi / 180
            hrand = hrand * rotx(rx) * roty(ry) * rotz(rz)
            return hrand

    # -------------------------------------------------------------
    # Program start:

    # Get the robot tool list
    tools = robot.Childs()

    # Get tools to calibrate (tools nambed with TCP_PREFIX):
    # Also, set visible the tools named with CHECK_COLLISION_NAME to check collisions

    sethidden = []
    print('Robot tools:')
    Htools = []
    ntools = len(tools)
    for i in range(ntools):
        tooli = tools[i]
        tooli_name = tooli.Name()
        if tooli_name.find(TCP_PREFIX) == 0:
            Htooli = tooli.PoseTool()
            print('Using %s to calibrate' % tooli_name)
            print(Htooli)
            Htools.append(Htooli)
        if tooli_name.find(CHECK_COLLISION_NAME) >= 0:
            print('Using TCP %s to check collision' % tooli_name)
            # Set the tool visible and remember if it was invisible to turn it off
            if not tooli.Visible():
                sethidden.append(tooli)
                tooli.setVisible(True)

    # Get objects to check collisions:
    all_objects = RDK.ItemList(ITEM_TYPE_OBJECT, True)
    nobjects = len(all_objects)
    for i in range(nobjects):
        objecti = RDK.Item(all_objects[i])
        objecti_name = objecti.Name()
        if objecti_name.find(CHECK_COLLISION_NAME) >= 0:
            print('Using object %s to check collision' % objecti_name)
            # Set the object visible and remember if it was hidden to turn it off
            if not objecti.Visible():
                sethidden.append(objecti)
                objecti.setVisible(True)

    ntools = len(Htools)
    if ntools <= 0:
        tooli = robot.AddTool(transl(100, 0, 100), TCP_PREFIX + ' 1')
        Htools.append(tooli.PoseTool())
        ntools = len(Htools)
        # raise Exception('No tools found with prefix: ' + TCP_PREFIX + '.\nRename the tools that you need to calibrate with the prefix: ' + TCP_PREFIX)

    Htracker_wrt_robot = invH(robot.PoseAbs()) * tracker.PoseAbs()
    ptracker = Htracker_wrt_robot[0:3, 3].tolist()

    # -----------------------------------------------------------------------
    print('Generating ' + repr(NMEASURES) + ' calibration/validation measurements.')
    JLIST = Mat(6, 0)
    JOINTS_REF = robot.JointsHome()

    #-----------
    robot.setJoints(JOINTS_REF)
    while CHECK_COLLISION and RDK.Collisions():
        RDK.Render()
        if ShowMessageYesNoCancel("The robot is in a collision state for the reference joints. Move the robot away from collisions.\n\nContinue?") is True:
            continue
        RDK.setCollisionActive(COLLISION_ON)
        quit()
    RDK.setCollisionActive(COLLISION_OFF)
    #-----------

    JOINTS_REF = robot.Joints()

    LAST_JOINTS = JOINTS_REF  #robot.Joints()
    TCPLIST = Mat(3, 0)

    i = -1
    id_measure = 0
    timeused = 0
    timeleft = -1
    tic()

    while id_measure < NMEASURES:
        i = i + 1
        idtool = id_measure % ntools
        Htool = Htools[idtool]
        ptool = Htool[0:3, 3]
        iHtool = invH(Htool)
        hi = randpose(robot, Htool, ptracker)
        print('Nmeasures: ' + repr(id_measure))
        print('Iteration: ' + repr(i))
        pose_flange = hi * iHtool
        print(pose_flange)
        ji = robot.SolveIK(pose_flange, JOINTS_REF)
        print('Testing Joints: ' + str(ji.list()))
        if not check_joints(ji):
            print('    Joint outside limits')
            continue
        if not check_pose(pose_flange):  #check_pose(hi):
            print('    Pose outside limits')
            continue

        # display potentially good configuration
        robot.setJoints(ji)
        if CHECK_COLLISION and RDK.Collisions():
            print('    End point is in a collision state %i' % i)
            continue
        if CHECK_WORKSPACE and not tool_object.IsInside(workspace_object):
            print('    Tool object outside measurement workspace %i' % i)
            continue
        if CHECK_COLLISION_MOVE and robot.MoveJ_Test(LAST_JOINTS, ji, CHECK_COLLISION_STEP) > 0:
            print('    MoveJ causes collision %i' % i)
            continue

        # robot.setJoints(ji) #this is made automatically by MoveJ_Collision
        LAST_JOINTS = ji
        JLIST = catH(JLIST, ji)
        TCPLIST = catH(TCPLIST, ptool)
        id_measure = id_measure + 1

        # Calculate time
        timeused = toc()
        timeavg = timeused / id_measure
        timeleft = (NMEASURES - id_measure) * timeavg
        print('Elapsed time      : %.1f sec ' % timeused)
        #print('Expected time left: %.1f sec  (average time x measure: %.1f sec)' % (timeleft, timeavg))
        message = 'Calculating measurement configurations. Expected time left: %.1f sec  (found %i/%i measurements)' % (timeleft, id_measure, NMEASURES)
        print(message)
        RDK.ShowMessage(message, False)

    NMEASURES_OK = id_measure
    SAVE_MAT = catV(JLIST, TCPLIST)

    if 'FILE_SAVE_PREFIX' in locals():
        strsave = RDK.getParam('PATH_OPENSTATION') + '/' + FILE_SAVE_PREFIX + repr(NMEASURES_OK) + '.txt'
        SAVE_MAT.save(strsave)
    #else:
    #    strsave = getSaveFile(RDK.getParam('PATH_OPENSTATION'))
    #    strsave = strsave.name
    #    SAVE_MAT.save(strsave)

    # -----------------------------------------------------------------------
    print(tr(JLIST))
    robot.ShowSequence(JLIST)
    RDK.ShowMessage('Calibration/validation sequence found', False)

    # Hide objects that we used to check collisions:
    nhide = len(sethidden)
    for i in range(nhide):
        sethidden[i].setVisible(False)

    # -----------------------------------------------------------------------
    calibitem = RDK.ItemUserPick("Select the calibration project", ITEM_TYPE_CALIBPROJECT)
    if not calibitem.Valid():
        raise Exception("No calibration project selected or available")
        return False

    if calib_targets is None:
        value = mbox('Do you want to use these targets for calibration or validation?', ('Calibration', 'CALIB_TARGETS'), ('Validation', 'VALID_TARGETS'))
    elif calib_targets:
        value = "CALIB_TARGETS"
    else:
        value = "VALID_TARGETS"

    calibitem.setValue(value, SAVE_MAT)

    RDK.ShowMessage('Done', False)

    #mbox('Done')
    # -----------------------------------------------------------------------

    #RDK.ShowSequence(Mat([[1, 10 ,10 ,10 ,10 ,10 ,10],[ 2, 20 ,20 ,20 ,20 ,20 ,20]]))
    return True


if __name__ == "__main__":
    CreateMeasurementsPoint()

--- Python program Prog11 ---
from robodk.robolink import *  # API to communicate with RoboDK
from robodk.robomath import *   # Robot toolbox
import robodk.robolinkutils as RDKutils
from robodk import robolink

DEBUG = False

# Link to RoboDK
RDK = Robolink()

ROBOT = RDK.ItemUserPick('Select a Robot', ITEM_TYPE_ROBOT)
FRAME = RDK.ItemUserPick('Reference Frame', ITEM_TYPE_FRAME)

if not ROBOT.Valid() or not FRAME.Valid():
    raise Exception("Select appropriate ROBOT and FRAME")

BASE = RDK.Item('UR10e Base', ITEM_TYPE_FRAME)
FRAMEPOSE = RDKutils.getPoseWrt(FRAME, BASE)  # frame pose with respect to robot base
TOOL = ROBOT.getLink(ITEM_TYPE_TOOL)
TOOLPOSE = RDKutils.getPoseWrt(TOOL, TOOL.Parent())  # tool pose with respect to robot flange

# Get all the holes as targets (only those with "H" in the name)
All_items = RDK.ItemList(ITEM_TYPE_TARGET)
RDK_items = [item for item in All_items if "H" in item.Name()]
print(f"Holes: {len(RDK_items)}")

RDK.setCollisionActive(COLLISION_OFF)

def print_xyzrpw(pose):
    x, y, z, rx, ry, rz = pose_2_xyzrpw(pose)
    print(x, y, z, rx, ry, rz)

class Hole:
    def __init__(self, pose, target):
        self.pose = pose
        self.target = target
        self.name = self.target.Name()
        self.split_position_rotation(pose)

    def split_position_rotation(self, pose):
        x, y, z, rx, ry, rz = pose_2_xyzrpw(pose)
        self.position = (x, y, z)
        # Get the z-axis direction (3rd column of the rotation matrix)
        self.rotation = pose[0:3, 2]
        zfacing1 = round(self.rotation.tolist()[0])
        zfacing2 = round(self.rotation.tolist()[1])
        zfacing3 = round(self.rotation.tolist()[2])
        self.rot_identifier = f"{zfacing1}_{zfacing2}_{zfacing3}"

class Face:
    def __init__(self, key):
        self.key = key
        self.get_midpoint(key)
        self.rotation = self.holes[0].rotation.tolist()
        self.offset_multiplier = self.rotation
        self.approaches = []  # Not used in the new functions

    def get_midpoint(self, key):
        # Retrieve all holes corresponding to this face
        self.holes = dic[key]
        x_values = [hole.position[0] for hole in self.holes]
        y_values = [hole.position[1] for hole in self.holes]
        z_values = [hole.position[2] for hole in self.holes]

        # Sort and compute the midpoint as the average of the min and max values
        x_values.sort()
        y_values.sort()
        z_values.sort()
        min_x, max_x = x_values[0], x_values[-1]
        min_y, max_y = y_values[0], y_values[-1]
        min_z, max_z = z_values[0], z_values[-1]

        mid_x = (min_x + max_x) / 2
        mid_y = (min_y + max_y) / 2
        mid_z = (min_z + max_z) / 2

        self.midpoint = (mid_x, mid_y, mid_z)

        # Use the first hole's pose as a template and update its translation to the midpoint
        self.ref_hole = self.holes[0]
        ref_pose = self.ref_hole.pose
        ref_pose[0, 3] = mid_x
        ref_pose[1, 3] = mid_y
        ref_pose[2, 3] = mid_z
        self.midpose = ref_pose

    def add_approaches(self, approach):
        self.approaches.append(approach)

# --- Process holes and group them into faces based on z-axis orientation ---
holes = []
dic = {}
faces = []

# Convert the target items into Hole objects
for item in RDK_items:
    hole = Hole(item.Pose(), item)
    holes.append(hole)

# Group holes with the same z-axis orientation (rounded)
for hole in holes:
    if hole.rot_identifier in dic:
        dic[hole.rot_identifier].append(hole)
    else:
        dic[hole.rot_identifier] = [hole]

# Create Face objects from the groups
for key in dic:
    face = Face(key)
    faces.append(face)

# --- NEW FUNCTION: Create face targets at the midpoint of each face ---
def create_face_targets():
    """
    For each computed face, create a new target in RoboDK at the face midpoint.
    """
    for i, face in enumerate(faces):
        face_target_name = f"Face_Target_{i}"
        existing_target = RDK.Item(face_target_name, ITEM_TYPE_TARGET)
        if existing_target.Valid():
            existing_target.Delete()
        face_target = RDK.AddTarget(face_target_name, FRAME, ROBOT)
        # face_target.setAsJointTarget() # joint target ?
        # face_target.setJoints(ROBOT.Joints())

        offset_transform = robomath.transl(0, 0, 0)
        adjusted_pose = face.midpose * offset_transform

        face_target.setPose(adjusted_pose)
        print(f"Created face target for face {i} at midpoint {face.midpoint}")

# --- NEW FUNCTION: Create a program for each face using MoveL commands ---
def create_face_programs():
    """
    For each face, generate a program that moves from the face target (approach target)
    to every hole target on that face using a MoveL command.
    Each move from the face target to a hole target is followed by a return move to the face target.
    """

    for i, face in enumerate(faces):
        face_target_name = f"Face_Target_{i}"
        face_target = RDK.Item(face_target_name, ITEM_TYPE_TARGET)
        prog_name = f"Program_Face_{i}"
        existing_prog = RDK.Item(prog_name, ITEM_TYPE_PROGRAM)
        if existing_prog.Valid():
            existing_prog.Delete()
        prog = RDK.AddProgram(prog_name, ROBOT)

        # Add a move to the face target as the starting (approach) move


        # For each hole in this face, add a MoveL to go to the hole target and then a MoveL back to the face target.
        for j, hole in enumerate(face.holes):  # Use enumerate to get the index 'j' of the hole

            # Construct the program names using f-strings
            program_to_call_2 = f'pickupToFaceTarget{i}'
            program_to_call_1 = f'FaceTarget{i}Topickup'

            if j == 0:
                prog.RunInstruction(program_to_call_2, robolink.INSTRUCTION_CALL_PROGRAM)

            prog.MoveL(face_target)
            prog.MoveL(hole.target)

            prog.RunInstruction('screw_in(20)', robolink.INSTRUCTION_CALL_PROGRAM)  # Tighten screw
            prog.RunInstruction('screw_out(0)', robolink.INSTRUCTION_CALL_PROGRAM)  # Release screwdriver

            prog.MoveL(face_target)

            prog.RunInstruction(program_to_call_1, robolink.INSTRUCTION_CALL_PROGRAM)

            # Check if it's NOT the last hole in the face
            if j < len(face.holes) - 1:

                prog.RunInstruction(program_to_call_2, robolink.INSTRUCTION_CALL_PROGRAM)

            print(f"Program {prog_name}: Added MoveL from approach target to hole {hole.name} and back.")

def addmainprogram():
    # set reference frame
    # set tcp

    prog_name = f"Program_Main"
    existing_prog = RDK.Item(prog_name, ITEM_TYPE_PROGRAM)
    if existing_prog.Valid():
        existing_prog.Delete()
    prog = RDK.AddProgram(prog_name, ROBOT)

    prog.setTool(RDK.ItemUserPick('Select tool', ITEM_TYPE_TOOL))
    prog.setFrame(RDK.ItemUserPick('Select frame', ITEM_TYPE_FRAME))

    # Voeg elke program toe aan een groot programma die met "program_face" begint

    for j in range(len(faces)):
        sub_prog_name = f"Program_Face_{j}"
        prog.RunInstruction(sub_prog_name)


def generate_pickup_links():
    # Define the name that is given in RoboDK for the pickup target
    pickup_target_name = "pickup"  # The name of the target in your RoboDK station

    # Get the actual RoboDK Item for the pickup target
    Target_Pickup_item = RDK.Item(pickup_target_name, ITEM_TYPE_TARGET)

    if not Target_Pickup_item.Valid():
        print(
            f"Error: Pickup target '{pickup_target_name}' not found in RoboDK station. Skipping pickup link generation.")
        return  # Exit the function if the pickup target doesn't exist

    # For every face, create 2 planned motions (programs)
    # One from Face_Target_i to 'pickup' target
    # One from 'pickup' target to Face_Target_i
    for i, face in enumerate(faces):  # Iterate through faces to get the numerical index 'i'
        # Get the name of the Face_Target for the current face
        face_target_name = f"Face_Target_{i}"

        # Define the names for the programs to be created by the plugin
        program_name_to_pickup = f"FaceTarget{i}Topickup"
        program_name_from_pickup = f"pickupToFaceTarget{i}" # Corrected: consistency with previous example

        # --- Check and delete existing "To Pickup" program ---
        existing_prog_to_pickup = RDK.Item(program_name_to_pickup, ITEM_TYPE_PROGRAM)
        if existing_prog_to_pickup.Valid():
            print(f"Deleting existing program: {program_name_to_pickup}")
            existing_prog_to_pickup.Delete()

